(****************************************************************************************************************************************************)
(***********                           start of the controlling of the message overlay and blocking of the visualisation                             ************)
(****************************************************************************************************************************************************)
(* Activate Error Message Overlay *)
	IF xActiveErrorMsg AND NOT(xEmergency) AND NOT(xNoAirPressure) AND NOT(xNodeFailCANOpen) THEN
		CASE iStepFunction OF
		(* Check *)
		1:	T_StartUp.T_State.xBlockChangeMovementVisu:=TRUE;	(* Lock the navigation of the visu *)
			(* Overlay Message Error *)
			T_VisuQVis.ptrT_ExchgParam^.T_SafetyCtrl.bStateMessageError:=1;
			T_VisuQVis.ptrT_ExchgParam^.T_SafetyCtrl.bStateMessageInfo:=0;
			T_VisuQVis.ptrT_ExchgParam^.T_SafetyCtrl.bStateMessageWarning:=0;
			T_VisuQVis.ptrT_ExchgParam^.T_SafetyCtrl.iMsgErrorLine1:=iMsgNumber;
			T_VisuQVis.ptrT_ExchgParam^.T_SafetyCtrl.iMsgErrorLine2:=iMsgNumber;
			T_VisuQVis.ptrT_ExchgParam^.T_SafetyCtrl.iMsgErrorLine3:=iMsgNumber;
			T_VisuQVis.ptrT_ExchgParam^.T_SafetyCtrl.iMsgErrorLine4:=iMsgNumber;
			T_VisuQVis.ptrT_ExchgParam^.T_SafetyCtrl.xConfirmMsgError:=FALSE;
			T_VisuQVis.ptrT_ExchgParam^.T_SafetyCtrl.xBlockVisuObject:=TRUE;
			(* next step *)
			iStepFunction:=10;
		10:	IF T_VisuQVis.ptrT_ExchgParam^.T_SafetyCtrl.xConfirmMsgError THEN
				T_VisuQVis.ptrT_ExchgParam^.T_SafetyCtrl.xBlockVisuObject:=FALSE;
				T_StartUp.T_State.xBlockChangeMovementVisu:=FALSE;	(* Unlock the navigation of the visu *)
				T_VisuQVis.ptrT_ExchgParam^.T_SafetyCtrl.bStateMessageError:=0;
				T_VisuQVis.ptrT_ExchgParam^.T_SafetyCtrl.xConfirmMsgError:=FALSE;
				T_StartUp.T_Ctrle.xDone:=TRUE;
				T_StartUp.T_Ctrle.xErr:=FALSE;
				T_StartUp.T_Ctrle.udiErrorID:=16#0;
				xActiveErrorMsg:=FALSE;
				(* next step *)
				iStepFunction:=1;
			END_IF;
		END_CASE;
	END_IF;

(* Acitvate Info Message Overlay *)
	IF xActiveInfoMsg AND NOT(xEmergency) AND NOT(xNoAirPressure) AND NOT(xNodeFailCANOpen) THEN
		CASE iStepFunction OF
		(* Check *)
		1:	T_StartUp.T_State.xBlockChangeMovementVisu:=TRUE;	(* Lock the navigation of the visu *)
			(* Overlay Message Error *)
			T_VisuQVis.ptrT_ExchgParam^.T_SafetyCtrl.bStateMessageError:=0;
			T_VisuQVis.ptrT_ExchgParam^.T_SafetyCtrl.bStateMessageInfo:=1;
			T_VisuQVis.ptrT_ExchgParam^.T_SafetyCtrl.bStateMessageWarning:=0;
			T_VisuQVis.ptrT_ExchgParam^.T_SafetyCtrl.iMsgInfoLine1:=iMsgNumber;
			T_VisuQVis.ptrT_ExchgParam^.T_SafetyCtrl.iMsgInfoLine2:=iMsgNumber;
			T_VisuQVis.ptrT_ExchgParam^.T_SafetyCtrl.iMsgInfoLine3:=iMsgNumber;
			T_VisuQVis.ptrT_ExchgParam^.T_SafetyCtrl.iMsgInfoLine4:=iMsgNumber;
			T_VisuQVis.ptrT_ExchgParam^.T_SafetyCtrl.xConfirmMsgInfo:=FALSE;
			T_VisuQVis.ptrT_ExchgParam^.T_SafetyCtrl.xBlockVisuObject:=TRUE;
			(* next step *)
			iStepFunction:=10;
		10:	IF T_VisuQVis.ptrT_ExchgParam^.T_SafetyCtrl.xConfirmMsgInfo THEN
				T_VisuQVis.ptrT_ExchgParam^.T_SafetyCtrl.xBlockVisuObject:=FALSE;
				T_StartUp.T_State.xBlockChangeMovementVisu:=FALSE;	(* Unlock the navigation of the visu *)
				T_VisuQVis.ptrT_ExchgParam^.T_SafetyCtrl.bStateMessageInfo:=0;
				T_VisuQVis.ptrT_ExchgParam^.T_SafetyCtrl.xConfirmMsgInfo:=FALSE;
				T_StartUp.T_Ctrle.xDone:=TRUE;
				T_StartUp.T_Ctrle.xErr:=FALSE;
				T_StartUp.T_Ctrle.udiErrorID:=16#0;
				xActiveInfoMsg:=FALSE;
				(* next step *)
				iStepFunction:=1;
			END_IF;
		END_CASE;
	END_IF;
(****************************************************************************************************************************************************)
(***********                           end of the controlling of the message overlay and blocking of the visualisation                             ************)
(****************************************************************************************************************************************************)

	IF T_StartUp.T_Ctrle.xSetSecurityStateON THEN
		IF NOT(xReadFirstTime) THEN
			xReadFirstTime:=TRUE;
			iStepFunctionON:=1;
			TONWaitSetSecStateON(IN:=FALSE);
		END_IF;
		CASE iStepFunctionON OF
		1:	T_TwinSafeCtrleOUT.xTwinSAFE_Run:=FALSE;	(* Stop TwinSafe Groupe *)
			QarxDigitalOutput[1]:=FALSE;	(* QxCtrlLampStartButton *)
			QarxDigitalOutput[2]:=FALSE;	(* QxCtrlLampStopButton *)
			QarxDigitalOutput[3]:=FALSE;	(* QxCtrlLampReleaseButton *)
			TONWaitSetSecStateON(IN:=FALSE);
			iStepFunctionON:=2;
		2:	TONWaitSetSecStateON(IN:=TRUE,PT:=T#50ms);
			IF TONWaitSetSecStateON.Q THEN
				TONWaitSetSecStateON(IN:=FALSE);
				iStepFunctionON:=3;
			END_IF;
		3:	T_TwinSafeCtrleOUT.xTwinSAFE_Run:=TRUE;	(* Start TwinSafe Groupe *)
			T_StartUp.T_Ctrle.xSetSecurityStateON:=FALSE;
			xReadFirstTime:=FALSE;
			TONWaitSetSecStateON(IN:=FALSE);
			iStepFunctionON:=1;
		END_CASE;
	ELSE
		xReadFirstTime:=FALSE;
	END_IF;

(****************************************************************************************************************************************************)
(***********                   start of the execution of an emergeny stop, missing of air or an axis communication error                  ************)
(****************************************************************************************************************************************************)
(* Emergency or air supply *)
	IF xEmergency OR xNoAirPressure OR xNodeFailCANOpen THEN
		CASE iStepFunction OF
		1:	xSetOutputDisable:=TRUE;
			T_NovRAM.T_Ctrle.xReset:=TRUE;
			T_StartUp.T_State.xBlockChangeMovementVisu:=TRUE;
			T_StartUp.T_Ctrle.iMsgNumber:=0;
			T_VisuQVis.ptrT_ExchgParam^.T_SafetyCtrl.iStateStartPage:=0;	(* No Text *)
			T_VisuQVis.ptrT_ExchgParam^.T_Visu.T_Level.iPwSystem:=999;	(* Releas System Level *)
			T_VisuQVis.ptrT_ExchgParam^.T_Visu.T_Level.iActLevel:=1;
			T_Process.xError:=FALSE;
			IF T_Process.xEnable AND NOT(T_Process.xEnd) AND ((T_Process.iFunctNr >= 50) AND (T_Process.iFunctNr <= 53)) THEN
				(* Prozess ist aktiv und wurde unterbrochen, daher müssen die letzten änderungen an den InfoProzess Parameter in den NovRam abgespeichert werden *)
				(* next step *)
				iStepFunction:=2;
			ELSE
				IF xProcessAbordet THEN
					xProcessAbordet:=FALSE;
					(* next step *)
					iStepFunction:=2;
				ELSE
					(* next step *)
					iStepFunction:=3;
				END_IF;
			END_IF;
		2:	IF NOT(T_NovRAM.T_Ctrle.xReset) AND T_NovRAM.T_Ctrle.xDone THEN
				iStepFunction:=3;
			END_IF;
		3:	IF NOT(T_NovRAM.T_Ctrle.xReset) AND T_NovRAM.T_Ctrle.xDone THEN
				T_VisuQVis.T_CtrleVisu.xReset:=TRUE;
				iStepFunction:=10;
			END_IF;
		(* waiting confirm *)
		10:	IF NOT(xSetOutputDisable) AND NOT(T_VisuQVis.T_CtrleVisu.xReset) THEN
				IF xNoAirPressure THEN
					(* next step *)
					iStepFunction:=60;
				END_IF;
				IF xEmergency THEN
					(* next step *)
					iStepFunction:=20;
				END_IF;
				IF xNodeFailCANOpen THEN
					(* next step *)
					iStepFunction:=80;
				END_IF;
			END_IF
		20:	(* Overlay Message Error *)
			T_VisuQVis.ptrT_ExchgParam^.T_SafetyCtrl.bStateMessageError:=1;
			T_VisuQVis.ptrT_ExchgParam^.T_SafetyCtrl.bStateMessageInfo:=0;
			T_VisuQVis.ptrT_ExchgParam^.T_SafetyCtrl.bStateMessageWarning:=0;
			T_VisuQVis.ptrT_ExchgParam^.T_SafetyCtrl.iMsgErrorLine1:=1;	(* EMERGENCY STOP BUTTON IS ACITVE! *)
			T_VisuQVis.ptrT_ExchgParam^.T_SafetyCtrl.iMsgErrorLine2:=1;	(* PLEASE RELEASE THIS BUTTON *)
			T_VisuQVis.ptrT_ExchgParam^.T_SafetyCtrl.iMsgErrorLine3:=1;	(* AND AFTER CONFIRM THIS MESSAGE *)
			T_VisuQVis.ptrT_ExchgParam^.T_SafetyCtrl.iMsgErrorLine4:=1;	(*  *)
			T_VisuQVis.ptrT_ExchgParam^.T_SafetyCtrl.xConfirmMsgError:=FALSE;
			T_VisuQVis.ptrT_ExchgParam^.T_SafetyCtrl.xBlockVisuObject:=TRUE;
			(* next step *)
			iStepFunction:=30;
		30:	IF T_VisuQVis.ptrT_ExchgParam^.T_SafetyCtrl.xConfirmMsgError THEN
				T_VisuQVis.ptrT_ExchgParam^.T_SafetyCtrl.xBlockVisuObject:=FALSE;
				T_VisuQVis.ptrT_ExchgParam^.T_SafetyCtrl.bStateMessageError:=0;
				T_VisuQVis.ptrT_ExchgParam^.T_SafetyCtrl.xConfirmMsgError:=FALSE;
				IF NOT(T_TwinSafeIn.IxEmergencyStopMachine) OR NOT(T_TwinSafeIn.IxEmergencyStopStuder) THEN
					(* next step *)
					iStepFunction:=20;
				ELSE
					(* next step *)
					iStepFunction:=90;
				END_IF;
			END_IF;
		60:	(* Overlay Message Error *)
			T_VisuQVis.ptrT_ExchgParam^.T_SafetyCtrl.bStateMessageError:=1;
			T_VisuQVis.ptrT_ExchgParam^.T_SafetyCtrl.bStateMessageInfo:=0;
			T_VisuQVis.ptrT_ExchgParam^.T_SafetyCtrl.bStateMessageWarning:=0;
			T_VisuQVis.ptrT_ExchgParam^.T_SafetyCtrl.iMsgErrorLine1:=2;	(* NO AIR PRESSURE! *)
			T_VisuQVis.ptrT_ExchgParam^.T_SafetyCtrl.iMsgErrorLine2:=2;	(* PLEASE ACTIVATE THE AIR PRESSURE *)
			T_VisuQVis.ptrT_ExchgParam^.T_SafetyCtrl.iMsgErrorLine3:=2;	(* AND AFTER CONFIRM THIS MESSAGE *)
			T_VisuQVis.ptrT_ExchgParam^.T_SafetyCtrl.iMsgErrorLine4:=2;	(*  *)
			T_VisuQVis.ptrT_ExchgParam^.T_SafetyCtrl.xConfirmMsgError:=FALSE;
			T_VisuQVis.ptrT_ExchgParam^.T_SafetyCtrl.xBlockVisuObject:=TRUE;
			FBErrorMessage(	diErrorNr:=7,		(* No Air Pressure *)
							T_ErrorList:=T_ErrorList);
			T_VisuQVis.ptrT_ExchgParam^.T_Visu.T_Message.sDynamicTextEnglish:=FBErrorMessage.sErrorTextEnglish;
			T_VisuQVis.ptrT_ExchgParam^.T_Visu.T_Message.sDynamicTextDeutsch:=FBErrorMessage.sErrorTextDeutsch;
			T_VisuQVis.ptrT_ExchgParam^.T_Visu.T_Message.sDynamicTextFrancais:=FBErrorMessage.sErrorTextFrancais;
			(* Safe the error *)
			T_VisuQVis.ptrT_ExchgParam^.T_SafetyCtrl.diSetForceErrorNr:=7;
			T_VisuQVis.ptrT_ExchgParam^.T_SafetyCtrl.xSetForceError:=TRUE;
			(* next step *)
			iStepFunction:=70;
		70:	IF T_VisuQVis.ptrT_ExchgParam^.T_SafetyCtrl.xConfirmMsgError THEN
				T_VisuQVis.ptrT_ExchgParam^.T_SafetyCtrl.xBlockVisuObject:=FALSE;
				T_VisuQVis.ptrT_ExchgParam^.T_SafetyCtrl.bStateMessageError:=0;
				T_VisuQVis.ptrT_ExchgParam^.T_SafetyCtrl.xConfirmMsgError:=FALSE;
				(* next step *)
				iStepFunction:=90;
			END_IF;
		80:	(* Overlay Message Error *)
			T_VisuQVis.ptrT_ExchgParam^.T_SafetyCtrl.bStateMessageError:=1;
			T_VisuQVis.ptrT_ExchgParam^.T_SafetyCtrl.bStateMessageInfo:=0;
			T_VisuQVis.ptrT_ExchgParam^.T_SafetyCtrl.bStateMessageWarning:=0;
			T_VisuQVis.ptrT_ExchgParam^.T_SafetyCtrl.iMsgErrorLine1:=21;	(* AT LEAST ONE CANOPEN CONTROLLER FAILED! *)
			T_VisuQVis.ptrT_ExchgParam^.T_SafetyCtrl.iMsgErrorLine2:=21;	(* PLEASE CHECK THE ECOSTEP AXIS *)
			T_VisuQVis.ptrT_ExchgParam^.T_SafetyCtrl.iMsgErrorLine3:=21;	(* AND CONFIRM THIS MESSAGE *)
			T_VisuQVis.ptrT_ExchgParam^.T_SafetyCtrl.iMsgErrorLine4:=21;	(*  *)
			T_VisuQVis.ptrT_ExchgParam^.T_SafetyCtrl.xConfirmMsgError:=FALSE;
			T_VisuQVis.ptrT_ExchgParam^.T_SafetyCtrl.xBlockVisuObject:=TRUE;
			FBErrorMessage(	diErrorNr:=6,		(* At least one Ecostep CANOpen Controller failed! *)
							T_ErrorList:=T_ErrorList);
			T_VisuQVis.ptrT_ExchgParam^.T_Visu.T_Message.sDynamicTextEnglish:=FBErrorMessage.sErrorTextEnglish;
			T_VisuQVis.ptrT_ExchgParam^.T_Visu.T_Message.sDynamicTextDeutsch:=FBErrorMessage.sErrorTextDeutsch;
			T_VisuQVis.ptrT_ExchgParam^.T_Visu.T_Message.sDynamicTextFrancais:=FBErrorMessage.sErrorTextFrancais;
			(* Safe the error *)
			T_VisuQVis.ptrT_ExchgParam^.T_SafetyCtrl.diSetForceErrorNr:=6;
			T_VisuQVis.ptrT_ExchgParam^.T_SafetyCtrl.xSetForceError:=TRUE;
			(* next step *)
			iStepFunction:=81;
		81:	IF T_VisuQVis.ptrT_ExchgParam^.T_SafetyCtrl.xConfirmMsgError THEN
				T_VisuQVis.ptrT_ExchgParam^.T_SafetyCtrl.xBlockVisuObject:=FALSE;
				T_VisuQVis.ptrT_ExchgParam^.T_SafetyCtrl.bStateMessageError:=0;
				T_VisuQVis.ptrT_ExchgParam^.T_SafetyCtrl.xConfirmMsgError:=FALSE;
				(* next step *)
				iStepFunction:=90;
			END_IF;
		(* end function or time out *)
		90:	xActiveErrorMsg:=FALSE;
			xActiveInfoMsg:=FALSE;
			T_StartUp.T_Ctrle.xDone:=TRUE;
			T_StartUp.T_Ctrle.xErr:=FALSE;
			T_StartUp.T_Ctrle.udiErrorID:=0;
			xEmergency:=FALSE;
			xNoAirPressure:=FALSE;
			xNodeFailCANOpen:=FALSE;
			xStartBooting:=TRUE;
			tTimeOutFunction:=T#0s;	(* deactivate the time out *)
			(* next step *)
			iStepFunction:=1;
		END_CASE
	END_IF;
(****************************************************************************************************************************************************)
(***********                   start of the execution of an emergeny stop, missing of air or an axis communication error                  ************)
(****************************************************************************************************************************************************)

(* Delete of the line error message *)
	IF xDeleteErrorMessage THEN
		xDeleteErrorMessage:=FALSE;
		FBInitErrorList(T_ErrorList:= T_ErrorList);	(* Init Static Text for Error List *)
		T_VisuQVis.ptrT_ExchgParam^.T_Visu.T_Message.sDynamicTextEnglish:='';
		T_VisuQVis.ptrT_ExchgParam^.T_Visu.T_Message.sDynamicTextDeutsch:='';
		T_VisuQVis.ptrT_ExchgParam^.T_Visu.T_Message.sDynamicTextFrancais:='';
		T_VisuQVis.ptrT_ExchgParam^.T_Visu.T_Message.iState:=0;
	END_IF;

(* Set Output disabled *)
	IF xSetOutputDisable THEN
		T_TwinSafeCtrleOUT.xTwinSAFE_Run:=FALSE;	(* Stop TwinSafe Groupe *)
		T_Process.xEnable:=FALSE;
		QarxDigitalOutput[1]:=FALSE;	(* QxCtrlLampStartButton *)
		QarxDigitalOutput[2]:=FALSE;	(* QxCtrlLampStopButton *)
		QarxDigitalOutput[3]:=FALSE;	(* QxCtrlLampReleaseButton *)
		QarxDigitalOutput[4]:=FALSE;	(* QxCtrlLampCurEcoButton *)
		T_Station.TControl.xEnable:=FALSE;
		T_VisuQVis.ptrT_ExchgParam^.T_Visu.iLoadingStartPage:=1;
		(* confirm *)
		xSetOutputDisable:=FALSE;
	END_IF
END_PROGRAM

(* POU PRG_PROCESS_LAYER4/FB_PROCESS/FB_InitErrorList, ST *)
FUNCTION_BLOCK FB_InitErrorList
VAR_INPUT
END_VAR
VAR_IN_OUT
	T_ErrorList:ST_ERROR_LIST;
END_VAR
VAR_OUTPUT
END_VAR
VAR
END_VAR
(****************************************************************************************************************************************************)
(***********                                    This Functionblock init all the error text in english, german and french                                       ************)
(****************************************************************************************************************************************************)
(* Static English Error List *)
T_ErrorList.asErrorListEnglish.T_LanguagList[1]:='Internal problem, should never appear';
T_ErrorList.asErrorListEnglish.T_LanguagList[2]:='Antivalence error of the motor encoder';
T_ErrorList.asErrorListEnglish.T_LanguagList[3]:='Encoder counter error, >+/- 4 inc';
T_ErrorList.asErrorListEnglish.T_LanguagList[4]:='Mster encoder X7 counter error, >+/- 4 inc';
T_ErrorList.asErrorListEnglish.T_LanguagList[5]:='Heat sink temperature to high (>80°)';
T_ErrorList.asErrorListEnglish.T_LanguagList[6]:='Low voltage (<18V) of the +24V logic supply';
T_ErrorList.asErrorListEnglish.T_LanguagList[7]:='High voltage X10 (>180V) of the motor power supply';
T_ErrorList.asErrorListEnglish.T_LanguagList[8]:='Low voltage X10 (<24V) of the motor power supply';
T_ErrorList.asErrorListEnglish.T_LanguagList[9]:='Short circuit in the motor phase A';
T_ErrorList.asErrorListEnglish.T_LanguagList[10]:='Short circuit in the motor phase B';
T_ErrorList.asErrorListEnglish.T_LanguagList[11]:='Short circuit of a digital output';
T_ErrorList.asErrorListEnglish.T_LanguagList[12]:='Digital input ENABLE going to low level';
T_ErrorList.asErrorListEnglish.T_LanguagList[13]:='Exceed max. countouring error';
T_ErrorList.asErrorListEnglish.T_LanguagList[14]:='Rotation speed to high, can not read encoder signal';
T_ErrorList.asErrorListEnglish.T_LanguagList[15]:='Can not find the commutation';
T_ErrorList.asErrorListEnglish.T_LanguagList[16]:='CAN-Communication broken by Node Guarding';
T_ErrorList.asErrorListEnglish.T_LanguagList[17]:='I^2t- Controlling triggered (current limit)';
T_ErrorList.asErrorListEnglish.T_LanguagList[18]:='ADS communication error';
T_ErrorList.asErrorListEnglish.T_LanguagList[19]:='Axis function time out error';
T_ErrorList.asErrorListEnglish.T_LanguagList[20]:='Axis function not implemented';
T_ErrorList.asErrorListEnglish.T_LanguagList[21]:='No HDD free resource, time out';
T_ErrorList.asErrorListEnglish.T_LanguagList[22]:='HDD error, no file found';
T_ErrorList.asErrorListEnglish.T_LanguagList[23]:='Axis Parameter File, wrong syntax';
T_ErrorList.asErrorListEnglish.T_LanguagList[24]:='Wrong Para Fct: Read Axis Parameter';
T_ErrorList.asErrorListEnglish.T_LanguagList[25]:='Limit End Switch Active';
T_ErrorList.asErrorListEnglish.T_LanguagList[26]:='PDOMapping Para File, wrong syntax';
T_ErrorList.asErrorListEnglish.T_LanguagList[27]:='Wrong Para Fct: Read PDOMapping Parameter';
T_ErrorList.asErrorListEnglish.T_LanguagList[28]:='No Axis Power Supply';
T_ErrorList.asErrorListEnglish.T_LanguagList[29]:='Wrong Para Fct: Move velocity';
T_ErrorList.asErrorListEnglish.T_LanguagList[30]:='Can not move, no power supply';
T_ErrorList.asErrorListEnglish.T_LanguagList[31]:='Wrong Para Fct: Move position absolute';
T_ErrorList.asErrorListEnglish.T_LanguagList[32]:='Wrong Para Fct: Move position relative';
T_ErrorList.asErrorListEnglish.T_LanguagList[33]:='Wrong Para Fct: Move referencing';
T_ErrorList.asErrorListEnglish.T_LanguagList[34]:='Fct CalcAnlgeRefIndex:Ref.Sensor not found';
T_ErrorList.asErrorListEnglish.T_LanguagList[35]:='Wrong Para Fct: Send Axis Parameter';
T_ErrorList.asErrorListEnglish.T_LanguagList[36]:='Wrong Para Fct: Send PDOMapping Parameter';
T_ErrorList.asErrorListEnglish.T_LanguagList[37]:='Wrong Para Fct: Master/Slave';
T_ErrorList.asErrorListEnglish.T_LanguagList[38]:='Axis general error';
T_ErrorList.asErrorListEnglish.T_LanguagList[39]:='ToolLeft: Wrong configuration or Axis missing';
T_ErrorList.asErrorListEnglish.T_LanguagList[40]:='ToolCenter: Wrong configuration or Axis missing';
T_ErrorList.asErrorListEnglish.T_LanguagList[41]:='ToolRight: Wrong configuration or Axis missing';
T_ErrorList.asErrorListEnglish.T_LanguagList[42]:='ToolFeeder: Wrong configuration or Axis missing';
T_ErrorList.asErrorListEnglish.T_LanguagList[43]:='GrindFeeder: Wrong configuration or Axis missing';
T_ErrorList.asErrorListEnglish.T_LanguagList[44]:='BoxId general error';
T_ErrorList.asErrorListEnglish.T_LanguagList[45]:='Cyl. Function not implemented';
T_ErrorList.asErrorListEnglish.T_LanguagList[46]:='Sensor down not active';
T_ErrorList.asErrorListEnglish.T_LanguagList[47]:='Sensor up not active';
T_ErrorList.asErrorListEnglish.T_LanguagList[48]:='Cyl. general error';
T_ErrorList.asErrorListEnglish.T_LanguagList[49]:='File for profile not found';
T_ErrorList.asErrorListEnglish.T_LanguagList[50]:='Profile file not found: ';
T_ErrorList.asErrorListEnglish.T_LanguagList[51]:='--> Load static default parameter';
T_ErrorList.asErrorListEnglish.T_LanguagList[52]:='Machine is not referenced';
T_ErrorList.asErrorListEnglish.T_LanguagList[53]:='Settled parameter for ToolLength is to long';
T_ErrorList.asErrorListEnglish.T_LanguagList[54]:='Settled parameter for ToolLength is to short';
T_ErrorList.asErrorListEnglish.T_LanguagList[55]:='Settled parameter for ToolDiameter is to big';
T_ErrorList.asErrorListEnglish.T_LanguagList[56]:='Settled parameter for ToolDiameter is to small';
T_ErrorList.asErrorListEnglish.T_LanguagList[57]:='Tool is not clamped';
T_ErrorList.asErrorListEnglish.T_LanguagList[58]:='ToolTension is not active';
T_ErrorList.asErrorListEnglish.T_LanguagList[59]:='ToolFeeeder is not on the StartPosition';
T_ErrorList.asErrorListEnglish.T_LanguagList[60]:='At least one Axis is busy';
T_ErrorList.asErrorListEnglish.T_LanguagList[61]:='Undefined Station error';
T_ErrorList.asErrorListEnglish.T_LanguagList[62]:='At least a passage of a section is not equal';
T_ErrorList.asErrorListEnglish.T_LanguagList[63]:='On the MicroWire it is not possible to Referencing';
T_ErrorList.asErrorListEnglish.T_LanguagList[64]:='Undefined Machine Error';
T_ErrorList.asErrorListEnglish.T_LanguagList[65]:='At least one Ecostep CANOpen Controller failed!';
T_ErrorList.asErrorListEnglish.T_LanguagList[66]:='No Air Pressure';
T_ErrorList.asErrorListEnglish.T_LanguagList[67]:='At least one settled diameter is bigger than ToolDiameter';
T_ErrorList.asErrorListEnglish.T_LanguagList[68]:='ToolTension is active';
T_ErrorList.asErrorListEnglish.T_LanguagList[69]:='';
T_ErrorList.asErrorListEnglish.T_LanguagList[70]:='';
T_ErrorList.asErrorListEnglish.T_LanguagList[71]:='';
T_ErrorList.asErrorListEnglish.T_LanguagList[72]:='';
T_ErrorList.asErrorListEnglish.T_LanguagList[73]:='';
T_ErrorList.asErrorListEnglish.T_LanguagList[74]:='';
T_ErrorList.asErrorListEnglish.T_LanguagList[75]:='';
T_ErrorList.asErrorListEnglish.T_LanguagList[76]:='';
T_ErrorList.asErrorListEnglish.T_LanguagList[77]:='';
T_ErrorList.asErrorListEnglish.T_LanguagList[78]:='';
T_ErrorList.asErrorListEnglish.T_LanguagList[79]:='';
T_ErrorList.asErrorListEnglish.T_LanguagList[80]:='';
T_ErrorList.asErrorListEnglish.T_LanguagList[81]:='';
T_ErrorList.asErrorListEnglish.T_LanguagList[82]:='';
T_ErrorList.asErrorListEnglish.T_LanguagList[83]:='';
T_ErrorList.asErrorListEnglish.T_LanguagList[84]:='';
T_ErrorList.asErrorListEnglish.T_LanguagList[85]:='';
T_ErrorList.asErrorListEnglish.T_LanguagList[86]:='';
T_ErrorList.asErrorListEnglish.T_LanguagList[87]:='';
T_ErrorList.asErrorListEnglish.T_LanguagList[88]:='';
T_ErrorList.asErrorListEnglish.T_LanguagList[89]:='';
T_ErrorList.asErrorListEnglish.T_LanguagList[90]:='';
T_ErrorList.asErrorListEnglish.T_LanguagList[91]:='';
T_ErrorList.asErrorListEnglish.T_LanguagList[92]:='';
T_ErrorList.asErrorListEnglish.T_LanguagList[93]:='';
T_ErrorList.asErrorListEnglish.T_LanguagList[94]:='';
T_ErrorList.asErrorListEnglish.T_LanguagList[95]:='';
T_ErrorList.asErrorListEnglish.T_LanguagList[96]:='';
T_ErrorList.asErrorListEnglish.T_LanguagList[97]:='';
T_ErrorList.asErrorListEnglish.T_LanguagList[98]:='';
T_ErrorList.asErrorListEnglish.T_LanguagList[99]:='';
T_ErrorList.asErrorListEnglish.T_LanguagList[100]:='';
T_ErrorList.asErrorListEnglish.T_LanguagList[101]:='';
T_ErrorList.asErrorListEnglish.T_LanguagList[102]:='';
T_ErrorList.asErrorListEnglish.T_LanguagList[103]:='';
T_ErrorList.asErrorListEnglish.T_LanguagList[104]:='';
T_ErrorList.asErrorListEnglish.T_LanguagList[105]:='';
T_ErrorList.asErrorListEnglish.T_LanguagList[106]:='';
T_ErrorList.asErrorListEnglish.T_LanguagList[107]:='';
T_ErrorList.asErrorListEnglish.T_LanguagList[108]:='';
T_ErrorList.asErrorListEnglish.T_LanguagList[109]:='';
T_ErrorList.asErrorListEnglish.T_LanguagList[110]:='';
T_ErrorList.asErrorListEnglish.T_LanguagList[111]:='';
T_ErrorList.asErrorListEnglish.T_LanguagList[112]:='';
T_ErrorList.asErrorListEnglish.T_LanguagList[113]:='';
T_ErrorList.asErrorListEnglish.T_LanguagList[114]:='';
T_ErrorList.asErrorListEnglish.T_LanguagList[115]:='';
T_ErrorList.asErrorListEnglish.T_LanguagList[116]:='';
T_ErrorList.asErrorListEnglish.T_LanguagList[117]:='';
T_ErrorList.asErrorListEnglish.T_LanguagList[118]:='';
T_ErrorList.asErrorListEnglish.T_LanguagList[119]:='';
T_ErrorList.asErrorListEnglish.T_LanguagList[120]:='';
T_ErrorList.asErrorListEnglish.T_LanguagList[121]:='';
T_ErrorList.asErrorListEnglish.T_LanguagList[122]:='';
T_ErrorList.asErrorListEnglish.T_LanguagList[123]:='';
T_ErrorList.asErrorListEnglish.T_LanguagList[124]:='';
T_ErrorList.asErrorListEnglish.T_LanguagList[125]:='';
T_ErrorList.asErrorListEnglish.T_LanguagList[126]:='';
T_ErrorList.asErrorListEnglish.T_LanguagList[127]:='';
T_ErrorList.asErrorListEnglish.T_LanguagList[128]:='';
T_ErrorList.asErrorListEnglish.T_LanguagList[129]:='';
T_ErrorList.asErrorListEnglish.T_LanguagList[130]:='';
T_ErrorList.asErrorListEnglish.T_LanguagList[131]:='';
T_ErrorList.asErrorListEnglish.T_LanguagList[132]:='';
T_ErrorList.asErrorListEnglish.T_LanguagList[133]:='';
T_ErrorList.asErrorListEnglish.T_LanguagList[134]:='';
T_ErrorList.asErrorListEnglish.T_LanguagList[135]:='';
T_ErrorList.asErrorListEnglish.T_LanguagList[136]:='';
T_ErrorList.asErrorListEnglish.T_LanguagList[137]:='';
T_ErrorList.asErrorListEnglish.T_LanguagList[138]:='';
T_ErrorList.asErrorListEnglish.T_LanguagList[139]:='';
T_ErrorList.asErrorListEnglish.T_LanguagList[140]:='';
T_ErrorList.asErrorListEnglish.T_LanguagList[141]:='';
T_ErrorList.asErrorListEnglish.T_LanguagList[142]:='';
T_ErrorList.asErrorListEnglish.T_LanguagList[143]:='';
T_ErrorList.asErrorListEnglish.T_LanguagList[144]:='';
T_ErrorList.asErrorListEnglish.T_LanguagList[145]:='';
T_ErrorList.asErrorListEnglish.T_LanguagList[146]:='';
T_ErrorList.asErrorListEnglish.T_LanguagList[147]:='';
T_ErrorList.asErrorListEnglish.T_LanguagList[148]:='';
T_ErrorList.asErrorListEnglish.T_LanguagList[149]:='';
T_ErrorList.asErrorListEnglish.T_LanguagList[150]:='';
T_ErrorList.asErrorListEnglish.T_LanguagList[151]:='';
T_ErrorList.asErrorListEnglish.T_LanguagList[152]:='';
T_ErrorList.asErrorListEnglish.T_LanguagList[153]:='';
T_ErrorList.asErrorListEnglish.T_LanguagList[154]:='';
T_ErrorList.asErrorListEnglish.T_LanguagList[155]:='';
T_ErrorList.asErrorListEnglish.T_LanguagList[156]:='';
T_ErrorList.asErrorListEnglish.T_LanguagList[157]:='';
T_ErrorList.asErrorListEnglish.T_LanguagList[158]:='';
T_ErrorList.asErrorListEnglish.T_LanguagList[159]:='';
T_ErrorList.asErrorListEnglish.T_LanguagList[160]:='';
T_ErrorList.asErrorListEnglish.T_LanguagList[161]:='';
T_ErrorList.asErrorListEnglish.T_LanguagList[162]:='';
T_ErrorList.asErrorListEnglish.T_LanguagList[163]:='';
T_ErrorList.asErrorListEnglish.T_LanguagList[164]:='';
T_ErrorList.asErrorListEnglish.T_LanguagList[165]:='';
T_ErrorList.asErrorListEnglish.T_LanguagList[166]:='';
T_ErrorList.asErrorListEnglish.T_LanguagList[167]:='';
T_ErrorList.asErrorListEnglish.T_LanguagList[168]:='';
T_ErrorList.asErrorListEnglish.T_LanguagList[169]:='';
T_ErrorList.asErrorListEnglish.T_LanguagList[170]:='';
T_ErrorList.asErrorListEnglish.T_LanguagList[171]:='';
T_ErrorList.asErrorListEnglish.T_LanguagList[172]:='';

(* Static Deutsch Error List *)
T_ErrorList.asErrorListDeutsch.T_LanguagList[1]:='Interne Ursache, darf niemals auftreten';
T_ErrorList.asErrorListDeutsch.T_LanguagList[2]:='Antivalenzfehler der Motorencodersignale';
T_ErrorList.asErrorListDeutsch.T_LanguagList[3]:='Encoder Zählfehler, >+/- 4 ink';
T_ErrorList.asErrorListDeutsch.T_LanguagList[4]:='Master Encoder X7 Zählfehler, >+/- 4 inc';
T_ErrorList.asErrorListDeutsch.T_LanguagList[5]:='Kühlkörpertemperatur zu hoch (> 80°)';
T_ErrorList.asErrorListDeutsch.T_LanguagList[6]:='Unterspannung (<18V) der +24V Logikversorgung';
T_ErrorList.asErrorListDeutsch.T_LanguagList[7]:='Überspannung X10 (>180V) der Leistungsversorgung';
T_ErrorList.asErrorListDeutsch.T_LanguagList[8]:='Unterspannung X10 (<24V) der Leistungsversorgung';
T_ErrorList.asErrorListDeutsch.T_LanguagList[9]:='Kurzschluss in Motorphase A';
T_ErrorList.asErrorListDeutsch.T_LanguagList[10]:='Kurzschluss in Motorphase B';
T_ErrorList.asErrorListDeutsch.T_LanguagList[11]:='Kurzschluss eines digitalen Ausgangs';
T_ErrorList.asErrorListDeutsch.T_LanguagList[12]:='Digital-Eingang ENABLE wurde auf Low-Pegel gesetzt';
T_ErrorList.asErrorListDeutsch.T_LanguagList[13]:='Max. Schleppfehler überschritten';
T_ErrorList.asErrorListDeutsch.T_LanguagList[14]:='Drehzahl zu hoch, Regler kann Encoder nicht mehr auslesen';
T_ErrorList.asErrorListDeutsch.T_LanguagList[15]:='Kommutierung nicht gefunden';
T_ErrorList.asErrorListDeutsch.T_LanguagList[16]:='CAN-Kommunikation unterbrochen bei Node Guarding';
T_ErrorList.asErrorListDeutsch.T_LanguagList[17]:='I^2t- Überwachung ausgelöst (Stromgrenze)';
T_ErrorList.asErrorListDeutsch.T_LanguagList[18]:='ADS communication error';
T_ErrorList.asErrorListDeutsch.T_LanguagList[19]:='Axis function time out error';
T_ErrorList.asErrorListDeutsch.T_LanguagList[20]:='Axis function not implemented';
T_ErrorList.asErrorListDeutsch.T_LanguagList[21]:='No HDD free resource, time out';
T_ErrorList.asErrorListDeutsch.T_LanguagList[22]:='HDD error, no file found';
T_ErrorList.asErrorListDeutsch.T_LanguagList[23]:='Axis Parameter File, wrong syntax';
T_ErrorList.asErrorListDeutsch.T_LanguagList[24]:='Wrong Para Fct: Read Axis Parameter';
T_ErrorList.asErrorListDeutsch.T_LanguagList[25]:='Limit End Switch Active';
T_ErrorList.asErrorListDeutsch.T_LanguagList[26]:='PDOMapping Para File, wrong syntax';
T_ErrorList.asErrorListDeutsch.T_LanguagList[27]:='Wrong Para Fct: Read PDOMapping Parameter';
T_ErrorList.asErrorListDeutsch.T_LanguagList[28]:='No Axis Power Supply';
T_ErrorList.asErrorListDeutsch.T_LanguagList[29]:='Wrong Para Fct: Move velocity';
T_ErrorList.asErrorListDeutsch.T_LanguagList[30]:='Can not move, no power supply';
T_ErrorList.asErrorListDeutsch.T_LanguagList[31]:='Wrong Para Fct: Move position absolute';
T_ErrorList.asErrorListDeutsch.T_LanguagList[32]:='Wrong Para Fct: Move position relative';
T_ErrorList.asErrorListDeutsch.T_LanguagList[33]:='Wrong Para Fct: Move referencing';
T_ErrorList.asErrorListDeutsch.T_LanguagList[34]:='Fct CalcAnlgeRefIndex:Ref.Sensor not found';
T_ErrorList.asErrorListDeutsch.T_LanguagList[35]:='Wrong Para Fct: Send Axis Parameter';
T_ErrorList.asErrorListDeutsch.T_LanguagList[36]:='Wrong Para Fct: Send PDOMapping Parameter';
T_ErrorList.asErrorListDeutsch.T_LanguagList[37]:='Wrong Para Fct: Master/Slave';
T_ErrorList.asErrorListDeutsch.T_LanguagList[38]:='Axis general error';
T_ErrorList.asErrorListDeutsch.T_LanguagList[39]:='ToolLeft: Wrong configuration or Axis missing';
T_ErrorList.asErrorListDeutsch.T_LanguagList[40]:='ToolCenter: Wrong configuration or Axis missing';
T_ErrorList.asErrorListDeutsch.T_LanguagList[41]:='ToolRight: Wrong configuration or Axis missing';
T_ErrorList.asErrorListDeutsch.T_LanguagList[42]:='ToolFeeder: Wrong configuration or Axis missing';
T_ErrorList.asErrorListDeutsch.T_LanguagList[43]:='GrindFeeder: Wrong configuration or Axis missing';
T_ErrorList.asErrorListDeutsch.T_LanguagList[44]:='BoxId general error';
T_ErrorList.asErrorListDeutsch.T_LanguagList[45]:='Cyl. Function not implemented';
T_ErrorList.asErrorListDeutsch.T_LanguagList[46]:='Sensor down not active';
T_ErrorList.asErrorListDeutsch.T_LanguagList[47]:='Sensor up not active';
T_ErrorList.asErrorListDeutsch.T_LanguagList[48]:='Cyl. general error';
T_ErrorList.asErrorListDeutsch.T_LanguagList[49]:='File for profile not found';
T_ErrorList.asErrorListDeutsch.T_LanguagList[50]:='Profile file not found: ';
T_ErrorList.asErrorListDeutsch.T_LanguagList[51]:='--> Load static default parameter';
T_ErrorList.asErrorListDeutsch.T_LanguagList[52]:='Machine is not referenced';
T_ErrorList.asErrorListDeutsch.T_LanguagList[53]:='Settled parameter for ToolLength is to long';
T_ErrorList.asErrorListDeutsch.T_LanguagList[54]:='Settled parameter for ToolLength is to short';
T_ErrorList.asErrorListDeutsch.T_LanguagList[55]:='Settled parameter for ToolDiameter is to big';
T_ErrorList.asErrorListDeutsch.T_LanguagList[56]:='Settled parameter for ToolDiameter is to small';
T_ErrorList.asErrorListDeutsch.T_LanguagList[57]:='Tool is not clamped';
T_ErrorList.asErrorListDeutsch.T_LanguagList[58]:='ToolTension is not active';
T_ErrorList.asErrorListDeutsch.T_LanguagList[59]:='ToolFeeeder is not on the StartPosition';
T_ErrorList.asErrorListDeutsch.T_LanguagList[60]:='At least one Axis is busy';
T_ErrorList.asErrorListDeutsch.T_LanguagList[61]:='Undefined Station error';
T_ErrorList.asErrorListDeutsch.T_LanguagList[62]:='At least a passage of a section is not equal';
T_ErrorList.asErrorListDeutsch.T_LanguagList[63]:='On the MicroWire it is not possible to Referencing';
T_ErrorList.asErrorListDeutsch.T_LanguagList[64]:='Undefined Machine Error';
T_ErrorList.asErrorListDeutsch.T_LanguagList[65]:='At least one Ecostep CANOpen Controller failed!';
T_ErrorList.asErrorListDeutsch.T_LanguagList[66]:='No Air Pressure';
T_ErrorList.asErrorListDeutsch.T_LanguagList[67]:='At least one settled diameter is bigger than ToolDiameter';
T_ErrorList.asErrorListDeutsch.T_LanguagList[68]:='ToolTension is active';
T_ErrorList.asErrorListDeutsch.T_LanguagList[69]:='';
T_ErrorList.asErrorListDeutsch.T_LanguagList[70]:='';
T_ErrorList.asErrorListDeutsch.T_LanguagList[71]:='';
T_ErrorList.asErrorListDeutsch.T_LanguagList[72]:='';
T_ErrorList.asErrorListDeutsch.T_LanguagList[73]:='';
T_ErrorList.asErrorListDeutsch.T_LanguagList[74]:='';
T_ErrorList.asErrorListDeutsch.T_LanguagList[75]:='';
T_ErrorList.asErrorListDeutsch.T_LanguagList[76]:='';
T_ErrorList.asErrorListDeutsch.T_LanguagList[77]:='';
T_ErrorList.asErrorListDeutsch.T_LanguagList[78]:='';
T_ErrorList.asErrorListDeutsch.T_LanguagList[79]:='';
T_ErrorList.asErrorListDeutsch.T_LanguagList[80]:='';
T_ErrorList.asErrorListDeutsch.T_LanguagList[81]:='';
T_ErrorList.asErrorListDeutsch.T_LanguagList[82]:='';
T_ErrorList.asErrorListDeutsch.T_LanguagList[83]:='';
T_ErrorList.asErrorListDeutsch.T_LanguagList[84]:='';
T_ErrorList.asErrorListDeutsch.T_LanguagList[85]:='';
T_ErrorList.asErrorListDeutsch.T_LanguagList[86]:='';
T_ErrorList.asErrorListDeutsch.T_LanguagList[87]:='';
T_ErrorList.asErrorListDeutsch.T_LanguagList[88]:='';
T_ErrorList.asErrorListDeutsch.T_LanguagList[89]:='';
T_ErrorList.asErrorListDeutsch.T_LanguagList[90]:='';
T_ErrorList.asErrorListDeutsch.T_LanguagList[91]:='';
T_ErrorList.asErrorListDeutsch.T_LanguagList[92]:='';
T_ErrorList.asErrorListDeutsch.T_LanguagList[93]:='';
T_ErrorList.asErrorListDeutsch.T_LanguagList[94]:='';
T_ErrorList.asErrorListDeutsch.T_LanguagList[95]:='';
T_ErrorList.asErrorListDeutsch.T_LanguagList[96]:='';
T_ErrorList.asErrorListDeutsch.T_LanguagList[97]:='';
T_ErrorList.asErrorListDeutsch.T_LanguagList[98]:='';
T_ErrorList.asErrorListDeutsch.T_LanguagList[99]:='';
T_ErrorList.asErrorListDeutsch.T_LanguagList[100]:='';
T_ErrorList.asErrorListDeutsch.T_LanguagList[101]:='';
T_ErrorList.asErrorListDeutsch.T_LanguagList[102]:='';
T_ErrorList.asErrorListDeutsch.T_LanguagList[103]:='';
T_ErrorList.asErrorListDeutsch.T_LanguagList[104]:='';
T_ErrorList.asErrorListDeutsch.T_LanguagList[105]:='';
T_ErrorList.asErrorListDeutsch.T_LanguagList[106]:='';
T_ErrorList.asErrorListDeutsch.T_LanguagList[107]:='';
T_ErrorList.asErrorListDeutsch.T_LanguagList[108]:='';
T_ErrorList.asErrorListDeutsch.T_LanguagList[109]:='';
T_ErrorList.asErrorListDeutsch.T_LanguagList[110]:='';
T_ErrorList.asErrorListDeutsch.T_LanguagList[111]:='';
T_ErrorList.asErrorListDeutsch.T_LanguagList[112]:='';
T_ErrorList.asErrorListDeutsch.T_LanguagList[113]:='';
T_ErrorList.asErrorListDeutsch.T_LanguagList[114]:='';
T_ErrorList.asErrorListDeutsch.T_LanguagList[115]:='';
T_ErrorList.asErrorListDeutsch.T_LanguagList[116]:='';
T_ErrorList.asErrorListDeutsch.T_LanguagList[117]:='';
T_ErrorList.asErrorListDeutsch.T_LanguagList[118]:='';
T_ErrorList.asErrorListDeutsch.T_LanguagList[119]:='';
T_ErrorList.asErrorListDeutsch.T_LanguagList[120]:='';
T_ErrorList.asErrorListDeutsch.T_LanguagList[121]:='';
T_ErrorList.asErrorListDeutsch.T_LanguagList[122]:='';
T_ErrorList.asErrorListDeutsch.T_LanguagList[123]:='';
T_ErrorList.asErrorListDeutsch.T_LanguagList[124]:='';
T_ErrorList.asErrorListDeutsch.T_LanguagList[125]:='';
T_ErrorList.asErrorListDeutsch.T_LanguagList[126]:='';
T_ErrorList.asErrorListDeutsch.T_LanguagList[127]:='';
T_ErrorList.asErrorListDeutsch.T_LanguagList[128]:='';
T_ErrorList.asErrorListDeutsch.T_LanguagList[129]:='';
T_ErrorList.asErrorListDeutsch.T_LanguagList[130]:='';
T_ErrorList.asErrorListDeutsch.T_LanguagList[131]:='';
T_ErrorList.asErrorListDeutsch.T_LanguagList[132]:='';
T_ErrorList.asErrorListDeutsch.T_LanguagList[133]:='';
T_ErrorList.asErrorListDeutsch.T_LanguagList[134]:='';
T_ErrorList.asErrorListDeutsch.T_LanguagList[135]:='';
T_ErrorList.asErrorListDeutsch.T_LanguagList[136]:='';
T_ErrorList.asErrorListDeutsch.T_LanguagList[137]:='';
T_ErrorList.asErrorListDeutsch.T_LanguagList[138]:='';
T_ErrorList.asErrorListDeutsch.T_LanguagList[139]:='';
T_ErrorList.asErrorListDeutsch.T_LanguagList[140]:='';
T_ErrorList.asErrorListDeutsch.T_LanguagList[141]:='';
T_ErrorList.asErrorListDeutsch.T_LanguagList[142]:='';
T_ErrorList.asErrorListDeutsch.T_LanguagList[143]:='';
T_ErrorList.asErrorListDeutsch.T_LanguagList[144]:='';
T_ErrorList.asErrorListDeutsch.T_LanguagList[145]:='';
T_ErrorList.asErrorListDeutsch.T_LanguagList[146]:='';
T_ErrorList.asErrorListDeutsch.T_LanguagList[147]:='';
T_ErrorList.asErrorListDeutsch.T_LanguagList[148]:='';
T_ErrorList.asErrorListDeutsch.T_LanguagList[149]:='';
T_ErrorList.asErrorListDeutsch.T_LanguagList[150]:='';
T_ErrorList.asErrorListDeutsch.T_LanguagList[151]:='';
T_ErrorList.asErrorListDeutsch.T_LanguagList[152]:='';
T_ErrorList.asErrorListDeutsch.T_LanguagList[153]:='';
T_ErrorList.asErrorListDeutsch.T_LanguagList[154]:='';
T_ErrorList.asErrorListDeutsch.T_LanguagList[155]:='';
T_ErrorList.asErrorListDeutsch.T_LanguagList[156]:='';
T_ErrorList.asErrorListDeutsch.T_LanguagList[157]:='';
T_ErrorList.asErrorListDeutsch.T_LanguagList[158]:='';
T_ErrorList.asErrorListDeutsch.T_LanguagList[159]:='';
T_ErrorList.asErrorListDeutsch.T_LanguagList[160]:='';
T_ErrorList.asErrorListDeutsch.T_LanguagList[161]:='';
T_ErrorList.asErrorListDeutsch.T_LanguagList[162]:='';
T_ErrorList.asErrorListDeutsch.T_LanguagList[163]:='';
T_ErrorList.asErrorListDeutsch.T_LanguagList[164]:='';
T_ErrorList.asErrorListDeutsch.T_LanguagList[165]:='';
T_ErrorList.asErrorListDeutsch.T_LanguagList[166]:='';
T_ErrorList.asErrorListDeutsch.T_LanguagList[167]:='';
T_ErrorList.asErrorListDeutsch.T_LanguagList[168]:='';
T_ErrorList.asErrorListDeutsch.T_LanguagList[169]:='';
T_ErrorList.asErrorListDeutsch.T_LanguagList[170]:='';
T_ErrorList.asErrorListDeutsch.T_LanguagList[171]:='';
T_ErrorList.asErrorListDeutsch.T_LanguagList[172]:='';

(* Static Francais Error List *)
T_ErrorList.asErrorListFrancais.T_LanguagList[1]:='Internal problem, should never appear';
T_ErrorList.asErrorListFrancais.T_LanguagList[2]:='Antivalence error of the motor encoder';
T_ErrorList.asErrorListFrancais.T_LanguagList[3]:='Encoder counter error, >+/- 4 inc';
T_ErrorList.asErrorListFrancais.T_LanguagList[4]:='Mster encoder X7 counter error, >+/- 4 inc';
T_ErrorList.asErrorListFrancais.T_LanguagList[5]:='Heat sink temperature to high (>80°)';
T_ErrorList.asErrorListFrancais.T_LanguagList[6]:='Low voltage (<18V) of the +24V logic supply';
T_ErrorList.asErrorListFrancais.T_LanguagList[7]:='High voltage X10 (>180V) of the motor power supply';
T_ErrorList.asErrorListFrancais.T_LanguagList[8]:='Low voltage X10 (<24V) of the motor power supply';
T_ErrorList.asErrorListFrancais.T_LanguagList[9]:='Short circuit in the motor phase A';
T_ErrorList.asErrorListFrancais.T_LanguagList[10]:='Short circuit in the motor phase B';
T_ErrorList.asErrorListFrancais.T_LanguagList[11]:='Short circuit of a digital output';
T_ErrorList.asErrorListFrancais.T_LanguagList[12]:='Digital input ENABLE going to low level';
T_ErrorList.asErrorListFrancais.T_LanguagList[13]:='Exceed max. countouring error ';
T_ErrorList.asErrorListFrancais.T_LanguagList[14]:='Rotation speed to high, can not read encoder signal';
T_ErrorList.asErrorListFrancais.T_LanguagList[15]:='Can not find the commutation';
T_ErrorList.asErrorListFrancais.T_LanguagList[16]:='CAN-Communication broken by Node Guarding';
T_ErrorList.asErrorListFrancais.T_LanguagList[17]:='I^2t- Controlling triggered (current limit)';
T_ErrorList.asErrorListFrancais.T_LanguagList[18]:='ADS communication error';
T_ErrorList.asErrorListFrancais.T_LanguagList[19]:='Axis function time out error';
T_ErrorList.asErrorListFrancais.T_LanguagList[20]:='Axis function not implemented';
T_ErrorList.asErrorListFrancais.T_LanguagList[21]:='No HDD free resource, time out';
T_ErrorList.asErrorListFrancais.T_LanguagList[22]:='HDD error, no file found';
T_ErrorList.asErrorListFrancais.T_LanguagList[23]:='Axis Parameter File, wrong syntax';
T_ErrorList.asErrorListFrancais.T_LanguagList[24]:='Wrong Para Fct: Read Axis Parameter';
T_ErrorList.asErrorListFrancais.T_LanguagList[25]:='Limit End Switch Active';
T_ErrorList.asErrorListFrancais.T_LanguagList[26]:='PDOMapping Para File, wrong syntax';
T_ErrorList.asErrorListFrancais.T_LanguagList[27]:='Wrong Para Fct: Read PDOMapping Parameter';
T_ErrorList.asErrorListFrancais.T_LanguagList[28]:='No Axis Power Supply';
T_ErrorList.asErrorListFrancais.T_LanguagList[29]:='Wrong Para Fct: Move velocity';
T_ErrorList.asErrorListFrancais.T_LanguagList[30]:='Can not move, no power supply';
T_ErrorList.asErrorListFrancais.T_LanguagList[31]:='Wrong Para Fct: Move position absolute';
T_ErrorList.asErrorListFrancais.T_LanguagList[32]:='Wrong Para Fct: Move position relative';
T_ErrorList.asErrorListFrancais.T_LanguagList[33]:='Wrong Para Fct: Move referencing';
T_ErrorList.asErrorListFrancais.T_LanguagList[34]:='Fct CalcAnlgeRefIndex:Ref.Sensor not found';
T_ErrorList.asErrorListFrancais.T_LanguagList[35]:='Wrong Para Fct: Send Axis Parameter';
T_ErrorList.asErrorListFrancais.T_LanguagList[36]:='Wrong Para Fct: Send PDOMapping Parameter';
T_ErrorList.asErrorListFrancais.T_LanguagList[37]:='Wrong Para Fct: Master/Slave';
T_ErrorList.asErrorListFrancais.T_LanguagList[38]:='Axis general error';
T_ErrorList.asErrorListFrancais.T_LanguagList[39]:='ToolLeft: Wrong configuration or Axis missing';
T_ErrorList.asErrorListFrancais.T_LanguagList[40]:='ToolCenter: Wrong configuration or Axis missing';
T_ErrorList.asErrorListFrancais.T_LanguagList[41]:='ToolRight: Wrong configuration or Axis missing';
T_ErrorList.asErrorListFrancais.T_LanguagList[42]:='ToolFeeder: Wrong configuration or Axis missing';
T_ErrorList.asErrorListFrancais.T_LanguagList[43]:='GrindFeeder: Wrong configuration or Axis missing';
T_ErrorList.asErrorListFrancais.T_LanguagList[44]:='BoxId general error';
T_ErrorList.asErrorListFrancais.T_LanguagList[45]:='Cyl. Function not implemented';
T_ErrorList.asErrorListFrancais.T_LanguagList[46]:='Sensor down not active';
T_ErrorList.asErrorListFrancais.T_LanguagList[47]:='Sensor up not active';
T_ErrorList.asErrorListFrancais.T_LanguagList[48]:='Cyl. general error';
T_ErrorList.asErrorListFrancais.T_LanguagList[49]:='File for profile not found';
T_ErrorList.asErrorListFrancais.T_LanguagList[50]:='Profile file not found: ';
T_ErrorList.asErrorListFrancais.T_LanguagList[51]:='--> Load static default parameter';
T_ErrorList.asErrorListFrancais.T_LanguagList[52]:='Machine is not referenced';
T_ErrorList.asErrorListFrancais.T_LanguagList[53]:='Settled parameter for ToolLength is to long';
T_ErrorList.asErrorListFrancais.T_LanguagList[54]:='Settled parameter for ToolLength is to short';
T_ErrorList.asErrorListFrancais.T_LanguagList[55]:='Settled parameter for ToolDiameter is to big';
T_ErrorList.asErrorListFrancais.T_LanguagList[56]:='Settled parameter for ToolDiameter is to small';
T_ErrorList.asErrorListFrancais.T_LanguagList[57]:='Tool is not clamped';
T_ErrorList.asErrorListFrancais.T_LanguagList[58]:='ToolTension is not active';
T_ErrorList.asErrorListFrancais.T_LanguagList[59]:='ToolFeeeder is not on the StartPosition';
T_ErrorList.asErrorListFrancais.T_LanguagList[60]:='At least one Axis is busy';
T_ErrorList.asErrorListFrancais.T_LanguagList[61]:='Undefined Station error';
T_ErrorList.asErrorListFrancais.T_LanguagList[62]:='At least a passage of a section is not equal';
T_ErrorList.asErrorListFrancais.T_LanguagList[63]:='On the MicroWire it is not possible to Referencing';
T_ErrorList.asErrorListFrancais.T_LanguagList[64]:='Undefined Machine Error';
T_ErrorList.asErrorListFrancais.T_LanguagList[65]:='At least one Ecostep CANOpen Controller failed!';
T_ErrorList.asErrorListFrancais.T_LanguagList[66]:='No Air Pressure';
T_ErrorList.asErrorListFrancais.T_LanguagList[67]:='At least one settled diameter is bigger than ToolDiameter';
T_ErrorList.asErrorListFrancais.T_LanguagList[68]:='ToolTension is active';
T_ErrorList.asErrorListFrancais.T_LanguagList[69]:='';
T_ErrorList.asErrorListFrancais.T_LanguagList[70]:='';
T_ErrorList.asErrorListFrancais.T_LanguagList[71]:='';
T_ErrorList.asErrorListFrancais.T_LanguagList[72]:='';
T_ErrorList.asErrorListFrancais.T_LanguagList[73]:='';
T_ErrorList.asErrorListFrancais.T_LanguagList[74]:='';
T_ErrorList.asErrorListFrancais.T_LanguagList[75]:='';
T_ErrorList.asErrorListFrancais.T_LanguagList[76]:='';
T_ErrorList.asErrorListFrancais.T_LanguagList[77]:='';
T_ErrorList.asErrorListFrancais.T_LanguagList[78]:='';
T_ErrorList.asErrorListFrancais.T_LanguagList[79]:='';
T_ErrorList.asErrorListFrancais.T_LanguagList[80]:='';
T_ErrorList.asErrorListFrancais.T_LanguagList[81]:='';
T_ErrorList.asErrorListFrancais.T_LanguagList[82]:='';
T_ErrorList.asErrorListFrancais.T_LanguagList[83]:='';
T_ErrorList.asErrorListFrancais.T_LanguagList[84]:='';
T_ErrorList.asErrorListFrancais.T_LanguagList[85]:='';
T_ErrorList.asErrorListFrancais.T_LanguagList[86]:='';
T_ErrorList.asErrorListFrancais.T_LanguagList[87]:='';
T_ErrorList.asErrorListFrancais.T_LanguagList[88]:='';
T_ErrorList.asErrorListFrancais.T_LanguagList[89]:='';
T_ErrorList.asErrorListFrancais.T_LanguagList[90]:='';
T_ErrorList.asErrorListFrancais.T_LanguagList[91]:='';
T_ErrorList.asErrorListFrancais.T_LanguagList[92]:='';
T_ErrorList.asErrorListFrancais.T_LanguagList[93]:='';
T_ErrorList.asErrorListFrancais.T_LanguagList[94]:='';
T_ErrorList.asErrorListFrancais.T_LanguagList[95]:='';
T_ErrorList.asErrorListFrancais.T_LanguagList[96]:='';
T_ErrorList.asErrorListFrancais.T_LanguagList[97]:='';
T_ErrorList.asErrorListFrancais.T_LanguagList[98]:='';
T_ErrorList.asErrorListFrancais.T_LanguagList[99]:='';
T_ErrorList.asErrorListFrancais.T_LanguagList[100]:='';
T_ErrorList.asErrorListFrancais.T_LanguagList[101]:='';
T_ErrorList.asErrorListFrancais.T_LanguagList[102]:='';
T_ErrorList.asErrorListFrancais.T_LanguagList[103]:='';
T_ErrorList.asErrorListFrancais.T_LanguagList[104]:='';
T_ErrorList.asErrorListFrancais.T_LanguagList[105]:='';
T_ErrorList.asErrorListFrancais.T_LanguagList[106]:='';
T_ErrorList.asErrorListFrancais.T_LanguagList[107]:='';
T_ErrorList.asErrorListFrancais.T_LanguagList[108]:='';
T_ErrorList.asErrorListFrancais.T_LanguagList[109]:='';
T_ErrorList.asErrorListFrancais.T_LanguagList[110]:='';
T_ErrorList.asErrorListFrancais.T_LanguagList[111]:='';
T_ErrorList.asErrorListFrancais.T_LanguagList[112]:='';
T_ErrorList.asErrorListFrancais.T_LanguagList[113]:='';
T_ErrorList.asErrorListFrancais.T_LanguagList[114]:='';
T_ErrorList.asErrorListFrancais.T_LanguagList[115]:='';
T_ErrorList.asErrorListFrancais.T_LanguagList[116]:='';
T_ErrorList.asErrorListFrancais.T_LanguagList[117]:='';
T_ErrorList.asErrorListFrancais.T_LanguagList[118]:='';
T_ErrorList.asErrorListFrancais.T_LanguagList[119]:='';
T_ErrorList.asErrorListFrancais.T_LanguagList[120]:='';
T_ErrorList.asErrorListFrancais.T_LanguagList[121]:='';
T_ErrorList.asErrorListFrancais.T_LanguagList[122]:='';
T_ErrorList.asErrorListFrancais.T_LanguagList[123]:='';
T_ErrorList.asErrorListFrancais.T_LanguagList[124]:='';
T_ErrorList.asErrorListFrancais.T_LanguagList[125]:='';
T_ErrorList.asErrorListFrancais.T_LanguagList[126]:='';
T_ErrorList.asErrorListFrancais.T_LanguagList[127]:='';
T_ErrorList.asErrorListFrancais.T_LanguagList[128]:='';
T_ErrorList.asErrorListFrancais.T_LanguagList[129]:='';
T_ErrorList.asErrorListFrancais.T_LanguagList[130]:='';
T_ErrorList.asErrorListFrancais.T_LanguagList[131]:='';
T_ErrorList.asErrorListFrancais.T_LanguagList[132]:='';
T_ErrorList.asErrorListFrancais.T_LanguagList[133]:='';
T_ErrorList.asErrorListFrancais.T_LanguagList[134]:='';
T_ErrorList.asErrorListFrancais.T_LanguagList[135]:='';
T_ErrorList.asErrorListFrancais.T_LanguagList[136]:='';
T_ErrorList.asErrorListFrancais.T_LanguagList[137]:='';
T_ErrorList.asErrorListFrancais.T_LanguagList[138]:='';
T_ErrorList.asErrorListFrancais.T_LanguagList[139]:='';
T_ErrorList.asErrorListFrancais.T_LanguagList[140]:='';
T_ErrorList.asErrorListFrancais.T_LanguagList[141]:='';
T_ErrorList.asErrorListFrancais.T_LanguagList[142]:='';
T_ErrorList.asErrorListFrancais.T_LanguagList[143]:='';
T_ErrorList.asErrorListFrancais.T_LanguagList[144]:='';
T_ErrorList.asErrorListFrancais.T_LanguagList[145]:='';
T_ErrorList.asErrorListFrancais.T_LanguagList[146]:='';
T_ErrorList.asErrorListFrancais.T_LanguagList[147]:='';
T_ErrorList.asErrorListFrancais.T_LanguagList[148]:='';
T_ErrorList.asErrorListFrancais.T_LanguagList[149]:='';
T_ErrorList.asErrorListFrancais.T_LanguagList[150]:='';
T_ErrorList.asErrorListFrancais.T_LanguagList[151]:='';
T_ErrorList.asErrorListFrancais.T_LanguagList[152]:='';
T_ErrorList.asErrorListFrancais.T_LanguagList[153]:='';
T_ErrorList.asErrorListFrancais.T_LanguagList[154]:='';
T_ErrorList.asErrorListFrancais.T_LanguagList[155]:='';
T_ErrorList.asErrorListFrancais.T_LanguagList[156]:='';
T_ErrorList.asErrorListFrancais.T_LanguagList[157]:='';
T_ErrorList.asErrorListFrancais.T_LanguagList[158]:='';
T_ErrorList.asErrorListFrancais.T_LanguagList[159]:='';
T_ErrorList.asErrorListFrancais.T_LanguagList[160]:='';
T_ErrorList.asErrorListFrancais.T_LanguagList[161]:='';
T_ErrorList.asErrorListFrancais.T_LanguagList[162]:='';
T_ErrorList.asErrorListFrancais.T_LanguagList[163]:='';
T_ErrorList.asErrorListFrancais.T_LanguagList[164]:='';
T_ErrorList.asErrorListFrancais.T_LanguagList[165]:='';
T_ErrorList.asErrorListFrancais.T_LanguagList[166]:='';
T_ErrorList.asErrorListFrancais.T_LanguagList[167]:='';
T_ErrorList.asErrorListFrancais.T_LanguagList[168]:='';
T_ErrorList.asErrorListFrancais.T_LanguagList[169]:='';
T_ErrorList.asErrorListFrancais.T_LanguagList[170]:='';
T_ErrorList.asErrorListFrancais.T_LanguagList[171]:='';
T_ErrorList.asErrorListFrancais.T_LanguagList[172]:='';
END_FUNCTION_BLOCK

(* POU GENERAL/FB_BIOSPARAMETER, ST *)
FUNCTION_BLOCK FB_BIOSPARAMETER
VAR_INPUT
	dwBIOSPasswordPage:DWORD;		(* Page number of the BIOS password page *)
	dwBIOSParameterPage:DWORD;		(* Page number of the BIOS parameter page *)
	T_TwinSafeOut:ST_TWINSAFE_OUT;	(* Output of the TwinSAFE components *)
END_VAR
VAR_IN_OUT
	T_Visu:ST_QVIS;						(* Data structure of the visualisation *)
	T_HDD:ST_HDD;						(* Data structure of the File Management *)
	T_NovRam : ST_NOVRAM;				(* Data structure of the NovRam *)
	T_CtrlePanel:ST_CTRLEPANEL;		(* Data structure of the ControlPanel *)
	T_DeviceID:ST_DEVICEID;				(* Data structure of the Device components *)
	T_BoxID:ST_BOXID;					(* Data structure of the components with the BoxId *)
	T_Profile:ST_PROFILE;				(* Data structure of the Profile management *)
END_VAR
VAR_OUTPUT
END_VAR
VAR
	TONShowMessage: TON;
	xChangeToBIOSPassword: BOOL;
	xChangeToBIOSParameter: BOOL;
	xSaveBIOSParameterToNovRAM: BOOL;
	xCopyBIOSParameter: BOOL;
	xReadFirstTimeParameter: BOOL;
	iStepSaveToNovRAM: INT;
	iStepReadFirstTimeParameter: INT;
	xCheckMsgBoxActive: BOOL;
(* Random *)
	fbGetCpuAccount:GETCPUCOUNTER;
	fbPwSystem:FBPW_SYSTEM;
	iPwSystem:INT;
	xNovRAMParaReaded: BOOL;
	xTmp: BOOL;
END_VAR
(****************************************************************************************************************************************************)
(***********     This Functionblock gives the possibility to set the bios parameter, with input a SystemLevel password     ************)
(****************************************************************************************************************************************************)
(* Managing BIOS Parameter on Startup *)
	IF (T_Visu.ptrT_ExchgParam^.T_Visu.T_Message.iStateBIOS <> 0) THEN
		TONShowMessage(IN:=TRUE,PT:=T#3s);
		IF TONShowMessage.Q THEN
			T_Visu.ptrT_ExchgParam^.T_Visu.T_Message.iStateBIOS:=0;
		END_IF;
	ELSE
		TONShowMessage(IN:=FALSE);
	END_IF;
	xCheckMsgBoxActive:=	(T_Visu.ptrT_ExchgParam^.T_SafetyCtrl.bStateMessageError <> 0) OR
							(T_Visu.ptrT_ExchgParam^.T_SafetyCtrl.bStateMessageInfo <> 0) OR
							(T_Visu.ptrT_ExchgParam^.T_SafetyCtrl.bStateMessageWarning <> 0);
	IF ((T_Visu.T_PlcParam.dwActualPage = 0) AND NOT(T_Visu.T_CtrleVisu.xExecute) AND T_Visu.T_CtrleVisu.xDone) OR xCheckMsgBoxActive THEN
		xChangeToBIOSPassword:=FALSE;
		xChangeToBIOSParameter:=FALSE;
		xSaveBIOSParameterToNovRAM:=FALSE;
		xCopyBIOSParameter:=FALSE;
		xReadFirstTimeParameter:=FALSE;
		iStepSaveToNovRAM:=1;
		iStepReadFirstTimeParameter:=1;
		T_Visu.ptrT_ExchgParam^.T_Visu.T_Message.iStateBIOS:=0;
		IF (T_Visu.ptrT_ExchgParam^.T_Config.iEditParam = DWORD_TO_INT(dwBIOSParameterPage)) THEN
			T_Visu.ptrT_ExchgParam^.T_Config.iEditParam:=0;
		END_IF;
	END_IF;
	IF (T_Visu.T_PlcParam.dwActualPage = dwBIOSPasswordPage) OR (T_Visu.T_PlcParam.dwActualPage = dwBIOSParameterPage) THEN
		IF (T_Visu.ptrT_ExchgParam^.T_SafetyCtrl.iStateStartPage = 2) THEN	(* check if external relase button has been pressed *)
			IF NOT(T_Visu.T_CtrleVisu.xExecute) AND T_Visu.T_CtrleVisu.xDone THEN
				T_Visu.T_PlcParam.dwSetNewPage:=0;
				T_Visu.T_CtrleVisu.iFunction:=1;
				T_Visu.T_CtrleVisu.xExecute:=TRUE;
			END_IF;
		END_IF;
	END_IF;
	(* check if the function button F1 is pressed-->if it is pressed the change to the BIOS password page *)
	IF NOT(xChangeToBIOSPassword) THEN
		IF (T_Visu.T_PlcParam.dwActualPage = 0) AND NOT(T_StartUp.T_State.xCompleted) THEN
			IF (T_Visu.ptrT_ExchgParam^.T_SafetyCtrl.iStateStartPage = 1) AND NOT(T_TwinSafeOut.QxContactor_K3) AND NOT(T_TwinSafeOut.QxContactor_K4) THEN
				IF T_Visu.ptrT_ExchgParam^.T_BtFunctionPanel.wActivBt = 16#1 THEN
					T_Visu.ptrT_ExchgParam^.T_BtFunctionPanel.wActivBt:=0;
					IF NOT(T_Visu.T_CtrleVisu.xExecute) AND T_Visu.T_CtrleVisu.xDone THEN
						T_Visu.ptrT_ExchgParam^.T_Visu.T_Message.iStateBIOS:=0;
						xChangeToBIOSPassword:=TRUE;
						T_Visu.T_PlcParam.dwSetNewPage:=dwBIOSPasswordPage;
						T_Visu.T_CtrleVisu.iFunction:=1;
						T_Visu.T_CtrleVisu.xExecute:=TRUE;
						fbGetCpuAccount;
						fbPwSystem(	dwCounter:=fbGetCpuAccount.fbGetCpuCounter.dwCpuCntHi+fbGetCpuAccount.fbGetCpuCounter.dwCpuCntLo,
									iRandom=>T_Visu.ptrT_ExchgParam^.T_Visu.T_Level.iRandom,
									iPwSystem=>iPwSystem);
					END_IF;
				END_IF;
			END_IF;
		END_IF;
	END_IF;
	(* check the settled password *)
	IF xChangeToBIOSPassword THEN
		IF (T_Visu.T_PlcParam.dwActualPage = dwBIOSPasswordPage) THEN
			IF T_Visu.ptrT_ExchgParam^.T_Visu.xKey_Escape THEN	(* ESC Button for exit and go to the Startpage *)
				T_Visu.ptrT_ExchgParam^.T_Visu.xKey_Escape:=FALSE;
				IF NOT(T_Visu.T_CtrleVisu.xExecute) AND T_Visu.T_CtrleVisu.xDone THEN
					xChangeToBIOSPassword:=FALSE;
					T_Visu.T_PlcParam.dwSetNewPage:=0;
					T_Visu.T_CtrleVisu.iFunction:=1;
					T_Visu.T_CtrleVisu.xExecute:=TRUE;
					T_Visu.ptrT_ExchgParam^.T_Visu.T_Level.iPwSystem:=999;
				END_IF;
			END_IF;
			IF (T_Visu.ptrT_ExchgParam^.T_Visu.T_Level.iPwSystem = iPwSystem) THEN
				T_Visu.ptrT_ExchgParam^.T_Visu.T_Message.iStateBIOS:=0;
				T_Visu.ptrT_ExchgParam^.T_Visu.T_Level.iPwSystem:=999;
				IF NOT(T_Visu.T_CtrleVisu.xExecute) AND T_Visu.T_CtrleVisu.xDone THEN
					xChangeToBIOSPassword:=FALSE;
					xChangeToBIOSParameter:=TRUE;
					T_Visu.T_PlcParam.dwSetNewPage:=dwBIOSParameterPage;
					T_Visu.T_CtrleVisu.iFunction:=1;
					T_Visu.T_CtrleVisu.xExecute:=TRUE;
					IF NOT(T_NovRam.T_Ctrle.xFirstRead) THEN
						xReadFirstTimeParameter:=TRUE;
					ELSE
						xCopyBIOSParameter:=TRUE;
					END_IF;
				END_IF;
			END_IF;
			IF (T_Visu.ptrT_ExchgParam^.T_Visu.T_Level.iPwSystem <> 999) THEN
				IF (T_Visu.ptrT_ExchgParam^.T_Visu.T_Level.iPwSystem <> iPwSystem) THEN
					T_Visu.ptrT_ExchgParam^.T_Visu.T_Message.iStateBIOS:=2;	(* Wrong password *)
					T_Visu.ptrT_ExchgParam^.T_Visu.T_Level.iPwSystem:=999;
				END_IF;
			END_IF;
		END_IF;
	END_IF;
	(* the edit parameterlist is now active *)
	IF xChangeToBIOSParameter AND NOT(xReadFirstTimeParameter) THEN
		T_Visu.ptrT_ExchgParam^.T_Config.iEditParam:=DWORD_TO_INT(dwBIOSParameterPage);
		IF (T_Visu.T_PlcParam.dwActualPage = dwBIOSParameterPage) AND NOT(xReadFirstTimeParameter) AND NOT(xSaveBIOSParameterToNovRAM) AND NOT(xCopyBIOSParameter) THEN
			IF T_Visu.ptrT_ExchgParam^.T_Visu.xKey_Escape THEN	(* ESC Button for exit and go to the Startpage *)
				T_Visu.ptrT_ExchgParam^.T_Visu.xKey_Escape:=FALSE;
				IF NOT(T_Visu.T_CtrleVisu.xExecute) AND T_Visu.T_CtrleVisu.xDone THEN
					xChangeToBIOSParameter:=FALSE;
					xSaveBIOSParameterToNovRAM:=FALSE;
					xCopyBIOSParameter:=TRUE;
					T_Visu.T_PlcParam.dwSetNewPage:=0;
					T_Visu.T_CtrleVisu.iFunction:=1;
					T_Visu.T_CtrleVisu.xExecute:=TRUE;
				END_IF;
			END_IF;
			IF (UDINT_TO_WORD(T_CtrlePanel.udiButton) = 16#200) AND NOT(xSaveBIOSParameterToNovRAM) THEN	(* Right Panel Button for save Parameter *)
				T_Visu.ptrT_ExchgParam^.T_Visu.T_Message.iStateBIOS:=1;	(* Parameter saved *)
				xSaveBIOSParameterToNovRAM:=TRUE;
				xCopyBIOSParameter:=FALSE;
				iStepSaveToNovRAM:=1;
			END_IF;
		END_IF;
	END_IF;
	(* save the settled parameter to the NovRam *)
	IF xSaveBIOSParameterToNovRAM THEN
		CASE iStepSaveToNovRAM OF
		1:	IF xNovRAMParaReaded THEN
				(* 30.11.2010 KFS: {	*)
				IF ( T_NovRam.T_Data.T_Standard.T_MachineConfig.rConfigMaxToolLength <> T_Visu.ptrT_ExchgParam^.T_StationCommon.rConfigMaxToolLength) THEN
					T_NovRam.T_Data.T_Standard.T_MachineConfig.rConfigMaxToolLengthOriginal:=0.0;
				END_IF;
				(* 30.11.2010 KFS:	}	*)
				T_NovRam.T_Data.T_Standard.T_MachineConfig.iConfigMachineType:=T_Visu.ptrT_ExchgParam^.T_StationCommon.iConfigMachineType;
				T_NovRam.T_Data.T_Standard.T_MachineConfig.iConfigAxisType:=T_Visu.ptrT_ExchgParam^.T_StationCommon.iConfigAxisType;
				T_NovRam.T_Data.T_Standard.T_MachineConfig.iConfigVisuNavigation:=T_Visu.ptrT_ExchgParam^.T_StationCommon.iConfigVisuNavigation;
				T_NovRam.T_Data.T_Standard.T_MachineConfig.rConfigMaxToolLength:=T_Visu.ptrT_ExchgParam^.T_StationCommon.rConfigMaxToolLength;
				T_NovRAM.T_Ctrle.iFunction:=2;
				T_NovRAM.T_Ctrle.xExecute:=TRUE;
				iStepSaveToNovRAM:=10;
			ELSE
				iStepSaveToNovRAM:=1;
				xSaveBIOSParameterToNovRAM:=FALSE;
			END_IF;
		10:	IF NOT(T_NovRAM.T_Ctrle.xExecute) AND T_NovRAM.T_Ctrle.xDone THEN
				iStepSaveToNovRAM:=1;
				xSaveBIOSParameterToNovRAM:=FALSE;
				T_Visu.T_CtrleVisu.xReset:=TRUE;	(* Exit the BIOS Parameter Page *)
			END_IF;
		END_CASE;
	END_IF;
	(* copy the NovRam config parameter to the visu structure *)
	IF xCopyBIOSParameter THEN
		IF xNovRAMParaReaded THEN
			T_Visu.ptrT_ExchgParam^.T_StationCommon.iConfigMachineType:=T_NovRam.T_Data.T_Standard.T_MachineConfig.iConfigMachineType;
			T_Visu.ptrT_ExchgParam^.T_StationCommon.iConfigAxisType:=T_NovRam.T_Data.T_Standard.T_MachineConfig.iConfigAxisType;
			T_Visu.ptrT_ExchgParam^.T_StationCommon.iConfigVisuNavigation:=T_NovRam.T_Data.T_Standard.T_MachineConfig.iConfigVisuNavigation;
			T_Visu.ptrT_ExchgParam^.T_StationCommon.rConfigMaxToolLength:=T_NovRam.T_Data.T_Standard.T_MachineConfig.rConfigMaxToolLength;
			T_Visu.ptrT_ExchgParam^.T_StationCommon.rConfigMaxToolLengthOriginal:=T_NovRam.T_Data.T_Standard.T_MachineConfig.rConfigMaxToolLengthOriginal;
			xCopyBIOSParameter:=FALSE;
		ELSE
			xCopyBIOSParameter:=FALSE;
		END_IF;
	END_IF;
	(* Init the Hardware for read the first time the parameter *)
	IF xReadFirstTimeParameter THEN
		CASE iStepReadFirstTimeParameter OF
		1:	T_HDD.T_Ctrle.xReset:=TRUE;
			T_DeviceID.T_Ctrle.xReset:=TRUE;
			T_BoxID.T_Ctrle.xReset:=TRUE;
			T_NovRAM.T_Ctrle.xReset:=TRUE;
			T_Profile.T_Ctrle.xReset:=TRUE;
			(* next step *)
			iStepReadFirstTimeParameter:=10;
			(* waiting reset confirmation *)
		10:	xTmp:=	T_HDD.T_Ctrle.xDone
					AND T_DeviceID.T_Ctrle.xDone
					AND T_NovRAM.T_Ctrle.xDone
					AND T_BoxID.T_Ctrle.xDone
					AND T_Profile.T_Ctrle.xDone;
			IF xTmp THEN  iStepReadFirstTimeParameter:=20; END_IF
		20:	(* PLC name *)
			T_DeviceID.T_CX1020.sDeviceName:='CX1000_PLC';
			(* feldbus name *)
			T_DeviceID.T_CANOpenMaster.sDeviceName:='CANOpenMaster';
			T_DeviceID.T_CANOpenMaster.xDeviceOption:=TRUE;
			T_DeviceID.T_LightbusMaster.sDeviceName:='LightbusMaster';
			T_DeviceID.T_LightbusMaster.xDeviceOption:=TRUE;
			(* NovRAM *)
			T_DeviceID.T_NovRAM.sDeviceName:='NovRAM';
			(* read device ID *)
			T_DeviceID.T_Ctrle.xExecute:=TRUE;
			(* next step *)
			iStepReadFirstTimeParameter:=30;
		(* waiting ID confirmation, Start BoxID *)
		30:	IF NOT(T_DeviceID.T_Ctrle.xExecute) AND T_DeviceID.T_Ctrle.xDone THEN iStepReadFirstTimeParameter:=40; END_IF
		(* waiting Box ID confirmation *)
		40:	IF NOT(T_BoxID.T_Ctrle.xExecute) AND T_BoxID.T_Ctrle.xDone THEN
				(* next step *)
				iStepReadFirstTimeParameter:=50;
			END_IF
		50:	T_NovRAM.T_Ctrle.iFunction:=1;
			T_NovRam.T_Ctrle.xBlockReadFirstTime:=TRUE;
			T_NovRAM.T_Ctrle.xExecute:=TRUE;
			iStepReadFirstTimeParameter:=60;
		60:	IF NOT(T_NovRAM.T_Ctrle.xExecute) AND T_NovRAM.T_Ctrle.xDone THEN
				xNovRAMParaReaded:=TRUE;
				T_Visu.ptrT_ExchgParam^.T_StationCommon.iConfigMachineType:=T_NovRam.T_Data.T_Standard.T_MachineConfig.iConfigMachineType;
				T_Visu.ptrT_ExchgParam^.T_StationCommon.iConfigAxisType:=T_NovRam.T_Data.T_Standard.T_MachineConfig.iConfigAxisType;
				T_Visu.ptrT_ExchgParam^.T_StationCommon.iConfigVisuNavigation:=T_NovRam.T_Data.T_Standard.T_MachineConfig.iConfigVisuNavigation;
				T_Visu.ptrT_ExchgParam^.T_StationCommon.rConfigMaxToolLength:=T_NovRam.T_Data.T_Standard.T_MachineConfig.rConfigMaxToolLength;
				T_Visu.ptrT_ExchgParam^.T_StationCommon.rConfigMaxToolLengthOriginal:=T_NovRam.T_Data.T_Standard.T_MachineConfig.rConfigMaxToolLengthOriginal;
				xReadFirstTimeParameter:=FALSE;
				iStepReadFirstTimeParameter:=1;
			END_IF;
		END_CASE;
	END_IF;
END_FUNCTION_BLOCK

(* POU PRG_VISU_LAYER5/FB_VISU/FBPW_SYSTEM, ST *)
FUNCTION_BLOCK FBPW_SYSTEM
VAR_INPUT
	dwCounter:DWORD;		(* number for generate the key *)
END_VAR
VAR_OUTPUT
	iRandom:INT;				(* generated key number for the password *)
	iPwSystem:INT;			(* level of the password *)
END_VAR
VAR
	i:INT;
	iCounter:INT;
	sTmp:STRING;
END_VAR
(****************************************************************************************************************************************************)
(***********                           This Functionblock is for the dynamic password, it generate a key number                                     ************)
(****************************************************************************************************************************************************)
(*
	dynamic System password
	ex : Counter=12345 => pw=55
	formul : 1+2+3+4+5 + 40 = 55
*)

(* Init. value *)
	iPwSystem:=0;
(* Convert value *)
	iCounter:=DWORD_TO_INT(dwCounter);
	IF iCounter<0 THEN iCounter:=iCounter*-1; END_IF
(* Set Random value *)
	iRandom:=iCounter;
	sTmp:=INT_TO_STRING(iCounter);
(* Set System pw *)
	FOR i:=0 TO LEN(sTmp)-1 DO
		iPwSystem:=iPwSystem+STRING_TO_INT(MID(sTmp,1,LEN(sTmp)-i));
		IF i=1 THEN iPwSystem:=iPwSystem+STRING_TO_INT(MID(sTmp,1,LEN(sTmp)-i))*10; END_IF
	END_FOR
END_FUNCTION_BLOCK

(* POU PRG_PROCESS_LAYER4/FB_PROCESS/FB_ErrorMessage, ST *)
FUNCTION_BLOCK FB_ErrorMessage
VAR_INPUT
	diErrorNr : DINT;				(* input of the error number *)
	T_ErrorList:ST_ERROR_LIST;	(* data structure of the errolist *)
END_VAR
VAR_OUTPUT
	sErrorTextEnglish : STRING(100);	(* give the error text in english *)
	sErrorTextDeutsch : STRING(100);	(* give the error text in german *)
	sErrorTextFrancais : STRING(100);	(* give the error text in french *)
END_VAR
VAR
	sTmpText1:STRING(100);
	sTmpText2:STRING(100);
	diTmpErrorNr:DINT;
	ptrErrorList: POINTER TO ST_LANGUAGE_LIST;
	iCounterLanguage: INT;
	sTmpErrorText : STRING(100);
	diTmpDeletePrefix: DINT;
END_VAR
(****************************************************************************************************************************************************)
(***********                     This Functionblock calculate all errors of the machine an set the follow errornumber                         ************)
(****************************************************************************************************************************************************)
ptrErrorList:=ADR(T_ErrorList.asErrorListEnglish);	(* pointer of the errorlist, default english *)
sErrorTextEnglish:='';
sErrorTextDeutsch:='';
sErrorTextFrancais:='';
sTmpText1:='';
diTmpErrorNr:=0;
diTmpDeletePrefix:=0;
(* detect the error of the hardware, station or process *)
IF (diErrorNr >= 1000000) AND (diErrorNr < 2000000) THEN
	diTmpDeletePrefix:=1000000;
	sTmpText1:='ToolLeft: ';
END_IF;
IF (diErrorNr >= 2000000) AND (diErrorNr < 3000000) THEN
	diTmpDeletePrefix:=2000000;
	sTmpText1:='ToolCenter: ';
END_IF;
IF (diErrorNr >= 3000000) AND (diErrorNr < 4000000) THEN
	diTmpDeletePrefix:=3000000;
	sTmpText1:='ToolRight: ';
END_IF;
IF (diErrorNr >= 4000000) AND (diErrorNr < 5000000) THEN
	diTmpDeletePrefix:=4000000;
	sTmpText1:='ToolFeeder: ';
END_IF;
IF (diErrorNr >= 5000000) AND (diErrorNr < 6000000) THEN
	diTmpDeletePrefix:=5000000;
	sTmpText1:='GrindFeeder: ';
END_IF;
IF (diErrorNr >= 6000000) AND (diErrorNr < 7000000) THEN
	diTmpDeletePrefix:=6000000;
	sTmpText1:='ToolTension: ';
END_IF;
IF (diErrorNr >= 7000000) AND (diErrorNr < 8000000) THEN
	diTmpDeletePrefix:=7000000;
	sTmpText1:='BoxId Err: ';
END_IF;
IF (diErrorNr >= 8000000) AND (diErrorNr < 9000000) THEN
	diTmpDeletePrefix:=8000000;
	sTmpText1:='Station Err: ';
END_IF;

FOR iCounterLanguage:=1 TO 3 DO
	sTmpText2:='';
	sTmpErrorText:='';
	(* set the pointer for the errorlist of the language english, german or french *)
	IF (iCounterLanguage = 1) THEN	ptrErrorList:=ADR(T_ErrorList.asErrorListEnglish); END_IF;
	IF (iCounterLanguage = 2) THEN	ptrErrorList:=ADR(T_ErrorList.asErrorListDeutsch); END_IF;
	IF (iCounterLanguage = 3) THEN	ptrErrorList:=ADR(T_ErrorList.asErrorListFrancais); END_IF;
	IF (diErrorNr >= 0) AND (diErrorNr < 1000000) THEN
		CASE diErrorNr OF
			1:			sTmpText2:=ptrErrorList^.T_LanguagList[52];		(* 'Machine is not referenced' *)
			2:			sTmpText2:=ptrErrorList^.T_LanguagList[57];		(* 'Tool is not clamped' *)
			3:			sTmpText2:=ptrErrorList^.T_LanguagList[58];		(* 'ToolTension is not active' *)
			4:			sTmpText2:=ptrErrorList^.T_LanguagList[59];		(* 'ToolFeeeder is not on the StartPosition' *)
			5:			sTmpText2:=ptrErrorList^.T_LanguagList[63];		(* 'On the MicroWire it is not possible to Referencing' *)
			6:			sTmpText2:=ptrErrorList^.T_LanguagList[65];		(* 'At least one Ecostep CANOpen Controller failed!' *)
			7:			sTmpText2:=ptrErrorList^.T_LanguagList[66];		(* 'No Air Pressure' *)
			16#F201:		sTmpText2:=ptrErrorList^.T_LanguagList[53];		(* 'Settled parameter for ToolLength is to long' *)
			16#F202:		sTmpText2:=ptrErrorList^.T_LanguagList[54];		(* 'Settled parameter for ToolLength is to short' *)
			16#F203:		sTmpText2:=ptrErrorList^.T_LanguagList[55];		(* 'Settled parameter for ToolDiameter is to big' *)
			16#F204:		sTmpText2:=ptrErrorList^.T_LanguagList[56];		(* 'Settled parameter for ToolDiameter is to small' *)
			16#F205:		sTmpText2:=ptrErrorList^.T_LanguagList[62];		(* 'At least a passage of a section is not equal' *)
			16#F206:		sTmpText2:=ptrErrorList^.T_LanguagList[67];		(* 'At least one settled diameter is bigger than ToolDiameter' *)
		ELSE
						sTmpText2:=ptrErrorList^.T_LanguagList[64];		(* 'Undefined Machine Error' *)
		END_CASE;
		sTmpErrorText:=CONCAT(sTmpText1,sTmpText2);
		IF (iCounterLanguage = 1) THEN sErrorTextEnglish:=sTmpErrorText;	END_IF;
		IF (iCounterLanguage = 2) THEN sErrorTextDeutsch:=sTmpErrorText;	END_IF;
		IF (iCounterLanguage = 3) THEN sErrorTextFrancais:=sTmpErrorText;	END_IF;
	ELSE
		IF (diErrorNr >= 1000000) AND (diErrorNr < 6000000) THEN
			diTmpErrorNr:=diErrorNr - diTmpDeletePrefix;
			CASE diTmpErrorNr OF
			16#F201:		sTmpText2:=ptrErrorList^.T_LanguagList[20];	(* 'Axis function not implemented' *)
			16#F202:		sTmpText2:=ptrErrorList^.T_LanguagList[21];	(* 'No HDD free resource, time out' *)
			16#F203:		sTmpText2:=ptrErrorList^.T_LanguagList[22];	(* 'HDD error, no file found' *)
			16#F204:		sTmpText2:=ptrErrorList^.T_LanguagList[23];	(* 'Axis Parameter File, wrong syntax' *)
			16#F205:		sTmpText2:=ptrErrorList^.T_LanguagList[26];	(* 'PDOMapping Para File, wrong syntax' *)
			16#F206:		sTmpText2:=ptrErrorList^.T_LanguagList[19];	(* 'Axis function time out error' *)
			16#F207:		sTmpText2:=ptrErrorList^.T_LanguagList[28];	(* 'No Axis Power Supply' *)
			16#F208:		sTmpText2:=ptrErrorList^.T_LanguagList[24];	(* 'Wrong Para Fct: Read Axis Parameter' *)
			16#F209:		sTmpText2:=ptrErrorList^.T_LanguagList[27];	(* 'Wrong Para Fct: Read PDOMapping Parameter' *)
			16#F20A:		sTmpText2:=ptrErrorList^.T_LanguagList[29];	(* 'Wrong Para Fct: Move velocity' *)
			16#F20B:		sTmpText2:=ptrErrorList^.T_LanguagList[31];	(* 'Wrong Para Fct: Move position absolute' *)
			16#F20C:		sTmpText2:=ptrErrorList^.T_LanguagList[32];	(* 'Wrong Para Fct: Move position relative' *)
			16#F20D:	sTmpText2:=ptrErrorList^.T_LanguagList[33];	(* 'Wrong Para Fct: Move referencing' *)
			16#F20E:		sTmpText2:=ptrErrorList^.T_LanguagList[35];	(* 'Wrong Para Fct: Send Axis Parameter' *)
			16#F20F:		sTmpText2:=ptrErrorList^.T_LanguagList[36];	(* 'Wrong Para Fct: Send PDOMapping Parameter' *)
			16#F210:		sTmpText2:=ptrErrorList^.T_LanguagList[37];	(* 'Wrong Para Fct: Master/Slave' *)
			16#F211:		sTmpText2:=ptrErrorList^.T_LanguagList[34];	(* 'Fct CalcAnlgeRefIndex:Ref.Sensor not found' *)
			16#F212:		sTmpText2:=ptrErrorList^.T_LanguagList[30];	(* 'Can not move, no power supply' *)
			16#F213:		sTmpText2:=ptrErrorList^.T_LanguagList[25];	(* 'Limit End Switch Active' *)
			16#F214:		sTmpText2:=ptrErrorList^.T_LanguagList[18];	(* 'ADS communication error' *)
			16#F801:		sTmpText2:=ptrErrorList^.T_LanguagList[1];	(* 'Internal problem, should never appear' *)
			16#F802:		sTmpText2:=ptrErrorList^.T_LanguagList[1];	(* 'Internal problem, should never appear' *)
			16#F803:		sTmpText2:=ptrErrorList^.T_LanguagList[2];	(* 'Antivalence error of the motor encoder' *)
			16#F804:		sTmpText2:=ptrErrorList^.T_LanguagList[3];	(* 'Encoder counter error, >+/- 4 inc' *)
			16#F805:		sTmpText2:=ptrErrorList^.T_LanguagList[4];	(* 'Master encoder X7 counter error, >+/- 4 inc' *)
			16#F806:		sTmpText2:=ptrErrorList^.T_LanguagList[5];	(* 'Heat sink temperature to high (>80°)' *)
			16#F807:		sTmpText2:=ptrErrorList^.T_LanguagList[6];	(* 'Low voltage (<18V) of the +24V logic supply' *)
			16#F808:		sTmpText2:=ptrErrorList^.T_LanguagList[7];	(* 'High voltage X10 (>180V) of the motor power supply' *)
			16#F809:		sTmpText2:=ptrErrorList^.T_LanguagList[8];	(* 'Low voltage X10 (<24V) of the motor power supply' *)
			16#F80A:		sTmpText2:=ptrErrorList^.T_LanguagList[9];	(* 'Short circuit in the motor phase A' *)
			16#F80B:		sTmpText2:=ptrErrorList^.T_LanguagList[10];	(* 'Short circuit in the motor phase B' *)
			16#F80C:		sTmpText2:=ptrErrorList^.T_LanguagList[11];	(* 'Short circuit of a digital output' *)
			16#F80D:	sTmpText2:=ptrErrorList^.T_LanguagList[12];	(* 'Digital input ENABLE going to low level' *)
			16#F80E:		sTmpText2:=ptrErrorList^.T_LanguagList[13];	(* 'Exceed max. countouring error ' *)
			16#F80F:		sTmpText2:=ptrErrorList^.T_LanguagList[14];	(* 'Rotation speed to high, can not read encoder signal' *)
			16#F810:		sTmpText2:=ptrErrorList^.T_LanguagList[15];	(* 'Can not find the commutation' *)
			16#F811:		sTmpText2:=ptrErrorList^.T_LanguagList[16];	(* 'CAN-Communication broken by Node Guarding' *)
			16#F812:		sTmpText2:=ptrErrorList^.T_LanguagList[17];	(* 'I^2t- Controlling triggered (current limit)' *)
			ELSE
						sTmpText2:=ptrErrorList^.T_LanguagList[38];	(* 'Axis general error' *)
			END_CASE;
		END_IF;
		IF (diErrorNr >= 6000000) AND (diErrorNr < 7000000) THEN
			diTmpErrorNr:=diErrorNr - diTmpDeletePrefix;
			CASE diTmpErrorNr OF
			16#F000:		sTmpText2:=ptrErrorList^.T_LanguagList[45];	(* 'Cyl. Function not implemented' *)
			16#F201:		sTmpText2:=ptrErrorList^.T_LanguagList[46];	(* 'Sensor down not active' *)
			16#F202:		sTmpText2:=ptrErrorList^.T_LanguagList[47];	(* 'Sensor up not active' *)
			ELSE
						sTmpText2:=ptrErrorList^.T_LanguagList[48];	(* 'Cyl. general error' *)
			END_CASE;
		END_IF;
		IF (diErrorNr >= 7000000) AND (diErrorNr < 8000000) THEN
			diTmpErrorNr:=diErrorNr - diTmpDeletePrefix;
			CASE diTmpErrorNr OF
			16#F201:		sTmpText2:=ptrErrorList^.T_LanguagList[39];	(* 'ToolLeft: Wrong configuration or Axis missing' *)
			16#F202:		sTmpText2:=ptrErrorList^.T_LanguagList[40];	(* 'ToolCenter: Wrong configuration or Axis missing' *)
			16#F203:		sTmpText2:=ptrErrorList^.T_LanguagList[41];	(* 'ToolRight: Wrong configuration or Axis missing' *)
			16#F204:		sTmpText2:=ptrErrorList^.T_LanguagList[42];	(* 'ToolFeeder: Wrong configuration or Axis missing' *)
			16#F205:		sTmpText2:=ptrErrorList^.T_LanguagList[43];	(* 'GrindFeeder: Wrong configuration or Axis missing' *)
			ELSE
						sTmpText2:=ptrErrorList^.T_LanguagList[44];	(* 'Cyl. general error' *)
			END_CASE;
		END_IF;
		IF (diErrorNr >= 8000000) AND (diErrorNr < 9000000) THEN
			diTmpErrorNr:=diErrorNr - diTmpDeletePrefix;
			CASE diTmpErrorNr OF
			1:			sTmpText2:=ptrErrorList^.T_LanguagList[60];	(* At least one Axis is busy *)
			2:			sTmpText2:=ptrErrorList^.T_LanguagList[68];
			ELSE
						sTmpText2:=ptrErrorList^.T_LanguagList[61];	(* Undefined Station error *)
			END_CASE;
		END_IF;
		IF (diErrorNr >= 10000000) AND (diErrorNr < 16000000) THEN
			diTmpErrorNr:=diErrorNr - diTmpDeletePrefix;
			CASE diTmpErrorNr OF
			16#F000:		sTmpText2:=ptrErrorList^.T_LanguagList[45];	(* 'Cyl. Function not implemented' *)
			16#F201:		sTmpText2:=ptrErrorList^.T_LanguagList[46];	(* 'Sensor down not active' *)
			16#F202:		sTmpText2:=ptrErrorList^.T_LanguagList[47];	(* 'Sensor up not active' *)
			ELSE
						sTmpText2:=ptrErrorList^.T_LanguagList[48];	(* 'Cyl. general error' *)
			END_CASE;
		END_IF;

		sTmpErrorText:=CONCAT(sTmpText1,sTmpText2);
		IF (iCounterLanguage = 1) THEN sErrorTextEnglish:=sTmpErrorText;	END_IF;
		IF (iCounterLanguage = 2) THEN sErrorTextDeutsch:=sTmpErrorText;	END_IF;
		IF (iCounterLanguage = 3) THEN sErrorTextFrancais:=sTmpErrorText;	END_IF;
	END_IF;
END_FOR;
END_FUNCTION_BLOCK

(* POU GENERAL/FB_CHECKACTIVEMOVEMENT, ST *)
FUNCTION_BLOCK FB_CHECKACTIVEMOVEMENT
VAR_INPUT
	T_TwinSafeOut:ST_TWINSAFE_OUT;		(* Output of the TwinSafe components *)
	xKeySwitch:BOOL;							(* Activation and deactivation of the key switch *)
	xBlockChecking:BOOL;						(* block the checking of the axis movement *)
END_VAR
VAR_IN_OUT
	xReset:BOOL;							(* Reset the FB *)
	T_Visu:ST_QVIS;							(* Data structure of the visualisation *)
	T_Station:ST_STATION;					(* Data structure of the station level *)
	T_Process : ST_PROCESS;				(* Data structure of the process level *)
END_VAR
VAR_OUTPUT
	xActiveSetupLevel: BOOL;					(* state of the setuplevel, if it is active *)
	xActiveProcess: BOOL;						(* state of a process if it is active *)
	xActiveStation: BOOL;						(* state of the stationlevel if it is active *)
	xActiveHWStation: BOOL;					(* state of the hardware of the station, if it is active *)
END_VAR
VAR
	xActivateOverlayMessage: BOOL;
	xDoNotCheckMovement: BOOL;
	FallingEdgeKeySwitchOff: F_TRIG;
	iStepSwitchMachineLevel: INT;
	TONWaitTimeStateMachine: TON;
	xPowerSupplyActive: BOOL;
	xTmp: BOOL;
	xStopAxisWithStationFunction: BOOL;
END_VAR
(****************************************************************************************************************************************************)
(*****        This Functionblock check the general movement of all axes. This will be need by change from the station level        ****)
(*****        to the machine level. If case of a change from the station level to the machine level and a axis move than the             ****)
(*****        movement will be stopp																			       ****)
(****************************************************************************************************************************************************)
(* Check Active movement and block visu if active *)
	xTmp:=	(T_Visu.ptrT_ExchgParam^.T_SafetyCtrl.bStateAutoGeometry = 2) OR
			(T_Visu.ptrT_ExchgParam^.T_SafetyCtrl.bStateAutoGroove = 2) OR
			(T_Visu.ptrT_ExchgParam^.T_SafetyCtrl.bStateReference = 2) OR
			(T_Visu.ptrT_ExchgParam^.T_SafetyCtrl.bStateToolCalibration = 2) OR
			(T_Visu.ptrT_ExchgParam^.T_SafetyCtrl.bStateToolTorque = 2) OR
			(T_Visu.ptrT_ExchgParam^.T_SafetyCtrl.bStateTeachInToolLeft = 2) OR
			(T_Visu.ptrT_ExchgParam^.T_SafetyCtrl.bStateTeachInToolCenter = 2) OR
			(T_Visu.ptrT_ExchgParam^.T_SafetyCtrl.bStateTeachInToolRight = 2) OR
			(T_Visu.ptrT_ExchgParam^.T_SafetyCtrl.bStateTeachInToolFeeder = 2) OR
			(T_Visu.ptrT_ExchgParam^.T_SafetyCtrl.bStateTeachInGrindFeeder = 2) OR
			(T_Visu.ptrT_ExchgParam^.T_StationCommon.iWireFeederRefIndexState = 2);
	IF xTmp THEN
		T_StartUp.T_State.xBlockVisuNavigation:=TRUE;	(* Lock the navigation of the visu *)
	END_IF;
	IF T_StartUp.T_State.xBlockVisuNavigation AND NOT(T_StartUp.T_State.xBlockChangeMovementVisu) AND NOT(T_Visu.ptrT_ExchgParam^.T_SafetyCtrl.xBlockVisuObject) AND NOT(xTmp) THEN
		T_StartUp.T_State.xBlockVisuNavigation:=FALSE;	(* Unlock the navigation of the visu *)
	END_IF;

(* Check Setup Level with active key switch and an active movement *)
	IF xReset THEN
		xReset:=FALSE;
		xActivateOverlayMessage:=FALSE;
	END_IF;
	IF NOT(xActivateOverlayMessage) THEN
		xActiveSetupLevel:=	(T_Visu.ptrT_ExchgParam^.T_Visu.bActivSpecialLayer <> 0) AND
							T_StartUp.T_State.xCompleted AND NOT(T_StartUp.T_State.xBlockChangeMovementVisu);
		xDoNotCheckMovement:=	NOT(T_Process.xEnd) AND NOT(T_Process.xError) AND ((T_Process.iFunctNr = 10) OR (T_Process.iFunctNr = 20) OR (T_Process.iFunctNr = 30));
		xActiveProcess:=		NOT(T_Process.xEnd) AND NOT(T_Process.xError) AND (T_Process.iFunctNr = 40);
		xActiveStation:=		NOT(T_Station.TControl.xEnd) AND NOT(T_Station.TControl.xError) AND NOT(xActiveProcess) AND NOT(xDoNotCheckMovement);
		xActiveHWStation:=	T_Station.TControl.xActiveMovement AND NOT(xActiveProcess) AND NOT(xActiveStation) AND NOT(xDoNotCheckMovement);
		(* check if the ToolTorque was activatet *)
		xStopAxisWithStationFunction:=FALSE;
		IF xActiveHWStation THEN
			IF (T_Visu.T_PlcParam.dwActualPage = 220) THEN
				xActiveHWStation:=FALSE;
				xStopAxisWithStationFunction:=TRUE;
			END_IF;
		END_IF;
	END_IF;
	FallingEdgeKeySwitchOff(CLK:=xKeySwitch);
	IF xActiveSetupLevel THEN
		IF FallingEdgeKeySwitchOff.Q THEN
			IF xActiveProcess OR xActiveStation OR xActiveHWStation OR xStopAxisWithStationFunction THEN
				xActivateOverlayMessage:=TRUE;
				iStepSwitchMachineLevel:=1;
			END_IF;
		END_IF;
	END_IF;
(*
	IF NOT(xBlockChecking) THEN
		xActivateOverlayMessage:= xActivateOverlayMessage AND NOT
								(T_Station.TControl.xSecurityCircuitOff OR T_Station.TControl.xSecurityCircuitOn);
	END_IF;
*)
	IF xActivateOverlayMessage THEN
		CASE iStepSwitchMachineLevel OF
		1:	TONWaitTimeStateMachine(IN:=FALSE);
			(* next step *)
			iStepSwitchMachineLevel:=10;
		10:	TONWaitTimeStateMachine(IN:=TRUE,PT:=T#150ms);
			IF TONWaitTimeStateMachine.Q THEN
				TONWaitTimeStateMachine(IN:=FALSE);
				(* next step *)
				iStepSwitchMachineLevel:=20;
			END_IF;
		20:	IF T_TwinSafeOut.QxContactor_K3 AND T_TwinSafeOut.QxContactor_K4 THEN
				xPowerSupplyActive:=TRUE;
				T_Visu.ptrT_ExchgParam^.T_Visu.T_Message.iState:=121;	(* Display message -> The Movement of the machine will be breaked! *)
				(* with switching off of the key switch the power supply is not switched off and the movement are still active *)
				IF xActiveProcess THEN
					T_Process.xStop:=TRUE;
					iStepSwitchMachineLevel:=30;
				END_IF;
				IF xActiveStation THEN
					T_Station.TControl.xStop:=TRUE;
					iStepSwitchMachineLevel:=40;
				END_IF;
				IF xActiveHWStation THEN
					iStepSwitchMachineLevel:=60;
				END_IF;
				IF xStopAxisWithStationFunction THEN
					iStepSwitchMachineLevel:=70;
				END_IF;
			ELSE
				(* with switching off of the key switch the power supply is switched off *)
				xPowerSupplyActive:=FALSE;
				(* next step *)
				iStepSwitchMachineLevel:=80;
			END_IF;
		30:	IF T_Process.xEnd THEN
				(* next step *)
				iStepSwitchMachineLevel:=80;
			END_IF;
			IF NOT(T_TwinSafeOut.QxContactor_K3) OR NOT(T_TwinSafeOut.QxContactor_K4) THEN
				xPowerSupplyActive:=FALSE;
				iStepSwitchMachineLevel:=80;
			END_IF;
			T_Visu.ptrT_ExchgParam^.T_Visu.T_Message.iState:=121;	(* Display message -> The Movement of the machine will be breaked! *)
		40:	IF T_Station.TControl.xEnd THEN
				(* next step *)
				T_Station.TControl.xStop:=FALSE;
				iStepSwitchMachineLevel:=60;
			END_IF;
			IF NOT(T_TwinSafeOut.QxContactor_K3) OR NOT(T_TwinSafeOut.QxContactor_K4) THEN
				xPowerSupplyActive:=FALSE;
				iStepSwitchMachineLevel:=80;
			END_IF;
			T_Visu.ptrT_ExchgParam^.T_Visu.T_Message.iState:=121;	(* Display message -> The Movement of the machine will be breaked! *)
		60:	IF T_Station.THardware.TAxisToolLeft.T_CtrleSingle.xDone AND NOT(T_Station.THardware.TAxisToolLeft.T_CtrleSingle.xErr) THEN
				T_Station.THardware.TAxisToolLeft.T_CtrleSingle.iFunction:=5;
				T_Station.THardware.TAxisToolLeft.T_CtrleSingle.xExecute:=TRUE;
			END_IF;
			IF NOT(T_Station.THardware.TAxisToolLeft.T_CtrleSingle.xDone) AND T_Station.THardware.TAxisToolLeft.T_CtrleSingle.xNotMoving AND NOT(T_Station.THardware.TAxisToolLeft.T_CtrleSingle.xErr) THEN
				T_Station.THardware.TAxisToolLeft.T_CtrleSingle.xReset:=TRUE;
			END_IF;
			IF T_Station.THardware.TAxisToolRight.T_CtrleSingle.xDone AND NOT(T_Station.THardware.TAxisToolRight.T_CtrleSingle.xErr) THEN
				T_Station.THardware.TAxisToolRight.T_CtrleSingle.iFunction:=5;
				T_Station.THardware.TAxisToolRight.T_CtrleSingle.xExecute:=TRUE;
			END_IF;
			IF NOT(T_Station.THardware.TAxisToolRight.T_CtrleSingle.xDone) AND T_Station.THardware.TAxisToolRight.T_CtrleSingle.xNotMoving AND NOT(T_Station.THardware.TAxisToolRight.T_CtrleSingle.xErr) THEN
				T_Station.THardware.TAxisToolRight.T_CtrleSingle.xReset:=TRUE;
			END_IF;
			IF T_Station.THardware.TAxisToolCenter.T_CtrleSingle.xDone AND NOT(T_Station.THardware.TAxisToolCenter.T_CtrleSingle.xErr) THEN
				T_Station.THardware.TAxisToolCenter.T_CtrleSingle.iFunction:=5;
				T_Station.THardware.TAxisToolCenter.T_CtrleSingle.xExecute:=TRUE;
			END_IF;
			IF NOT(T_Station.THardware.TAxisToolCenter.T_CtrleSingle.xDone) AND T_Station.THardware.TAxisToolCenter.T_CtrleSingle.xNotMoving AND NOT(T_Station.THardware.TAxisToolCenter.T_CtrleSingle.xErr) THEN
				T_Station.THardware.TAxisToolCenter.T_CtrleSingle.xReset:=TRUE;
			END_IF;
			IF T_Station.THardware.TAxisToolFeeder.T_CtrleSingle.xDone AND NOT(T_Station.THardware.TAxisToolFeeder.T_CtrleSingle.xErr) THEN
				T_Station.THardware.TAxisToolFeeder.T_CtrleSingle.iFunction:=5;
				T_Station.THardware.TAxisToolFeeder.T_CtrleSingle.xExecute:=TRUE;
			END_IF;
			IF NOT(T_Station.THardware.TAxisToolFeeder.T_CtrleSingle.xDone) AND NOT(T_Station.THardware.TAxisToolFeeder.T_CtrleSingle.xNotMoving) AND NOT(T_Station.THardware.TAxisToolFeeder.T_CtrleSingle.xErr) THEN
				T_Station.THardware.TAxisToolFeeder.T_CtrleSingle.iFunction:=5;
				T_Station.THardware.TAxisToolFeeder.T_CtrleSingle.xExecute:=TRUE;
			END_IF;
			IF NOT(T_Station.THardware.TAxisToolFeeder.T_CtrleSingle.xDone) AND T_Station.THardware.TAxisToolFeeder.T_CtrleSingle.xNotMoving AND NOT(T_Station.THardware.TAxisToolFeeder.T_CtrleSingle.xErr) THEN
				T_Station.THardware.TAxisToolFeeder.T_CtrleSingle.xReset:=TRUE;
			END_IF;
			IF T_Station.THardware.TAxisGrindFeeder.T_CtrleSingle.xDone AND NOT(T_Station.THardware.TAxisGrindFeeder.T_CtrleSingle.xErr) THEN
				T_Station.THardware.TAxisGrindFeeder.T_CtrleSingle.iFunction:=5;
				T_Station.THardware.TAxisGrindFeeder.T_CtrleSingle.xExecute:=TRUE;
			END_IF;
			IF NOT(T_Station.THardware.TAxisGrindFeeder.T_CtrleSingle.xDone) AND NOT(T_Station.THardware.TAxisGrindFeeder.T_CtrleSingle.xNotMoving) AND NOT(T_Station.THardware.TAxisGrindFeeder.T_CtrleSingle.xErr) THEN
				T_Station.THardware.TAxisGrindFeeder.T_CtrleSingle.iFunction:=5;
				T_Station.THardware.TAxisGrindFeeder.T_CtrleSingle.xExecute:=TRUE;
			END_IF;
			IF NOT(T_Station.THardware.TAxisGrindFeeder.T_CtrleSingle.xDone) AND T_Station.THardware.TAxisGrindFeeder.T_CtrleSingle.xNotMoving AND NOT(T_Station.THardware.TAxisGrindFeeder.T_CtrleSingle.xErr) THEN
				T_Station.THardware.TAxisGrindFeeder.T_CtrleSingle.xReset:=TRUE;
			END_IF;
			IF NOT(T_Station.THardware.TCylToolTension.T_CtrleCyl.xDone) THEN T_Station.THardware.TCylToolTension.T_CtrleCyl.xReset:=TRUE; END_IF;
			T_Visu.ptrT_ExchgParam^.T_Visu.T_Message.iState:=121;	(* Display message -> The Movement of the machine will be breaked! *)
			(* next step *)
			iStepSwitchMachineLevel:=80;
		70:	IF T_Station.TControl.xEnd THEN
				(* next step *)
				T_Station.TControl.iFunctNr:=3;
				T_Station.TControl.xStart:=TRUE;
				iStepSwitchMachineLevel:=71;
			END_IF;
			IF NOT(T_TwinSafeOut.QxContactor_K3) OR NOT(T_TwinSafeOut.QxContactor_K4) THEN
				xPowerSupplyActive:=FALSE;
				iStepSwitchMachineLevel:=80;
			END_IF;
			T_Visu.ptrT_ExchgParam^.T_Visu.T_Message.iState:=121;	(* Display message -> The Movement of the machine will be breaked! *)
		71:	IF NOT(T_Station.TControl.xStart) AND T_Station.TControl.xEnd THEN
				(* next step *)
				iStepSwitchMachineLevel:=80;
			END_IF;
			IF NOT(T_TwinSafeOut.QxContactor_K3) OR NOT(T_TwinSafeOut.QxContactor_K4) THEN
				xPowerSupplyActive:=FALSE;
				iStepSwitchMachineLevel:=80;
			END_IF;
		80:	IF NOT(T_Visu.T_CtrleVisu.xExecute) AND T_Visu.T_CtrleVisu.xDone THEN
				T_Visu.ptrT_ExchgParam^.T_Visu.T_Message.iState:=0;
				T_Visu.ptrT_ExchgParam^.T_Visu.bActivSpecialLayer:=0;
				T_Visu.ptrT_ExchgParam^.T_TouchScreenBtPanel.iStateBtLeft:=0;
				T_Visu.ptrT_ExchgParam^.T_TouchScreenNavPanel.wState:=1;
				T_Visu.T_PlcParam.dwSetNewPage:=16#A;	(* Main Page wird aufgerufen *)
				T_Visu.T_CtrleVisu.iFunction:=1;
				T_Visu.T_CtrleVisu.xExecute:=TRUE;
				iStepSwitchMachineLevel:=90;
			END_IF;
		90:	IF NOT(T_Visu.T_CtrleVisu.xExecute) AND T_Visu.T_CtrleVisu.xDone THEN
				T_StartUp.T_State.xBlockChangeMovementVisu:=TRUE;	(* Lock the navigation of the visu *)
				T_Visu.ptrT_ExchgParam^.T_SafetyCtrl.xBlockVisuObject:=TRUE;
				T_StartUp.T_State.xBlockVisuNavigation:=FALSE;	(* Unlock the navigation of the visu *)
				T_Visu.ptrT_ExchgParam^.T_SafetyCtrl.bStateAutoGeometry:=1;
				T_Visu.ptrT_ExchgParam^.T_SafetyCtrl.bStateAutoGroove:=1;
				T_Visu.ptrT_ExchgParam^.T_SafetyCtrl.bStateReference:=1;
				T_Visu.ptrT_ExchgParam^.T_SafetyCtrl.bStateToolCalibration:=1;
				T_Visu.ptrT_ExchgParam^.T_SafetyCtrl.bStateToolTorque:=1;
				T_Visu.ptrT_ExchgParam^.T_SafetyCtrl.bStateTeachInToolLeft:=1;
				T_Visu.ptrT_ExchgParam^.T_SafetyCtrl.bStateTeachInToolCenter:=1;
				T_Visu.ptrT_ExchgParam^.T_SafetyCtrl.bStateTeachInToolRight:=1;
				T_Visu.ptrT_ExchgParam^.T_SafetyCtrl.bStateTeachInToolFeeder:=1;
				T_Visu.ptrT_ExchgParam^.T_SafetyCtrl.bStateTeachInGrindFeeder:=1;
				T_Visu.ptrT_ExchgParam^.T_StationCommon.iWireFeederRefIndexState:=1;
				(* Overlay Message Error *)
				T_Visu.ptrT_ExchgParam^.T_SafetyCtrl.bStateMessageError:=1;
				T_Visu.ptrT_ExchgParam^.T_SafetyCtrl.bStateMessageInfo:=0;
				T_Visu.ptrT_ExchgParam^.T_SafetyCtrl.bStateMessageWarning:=0;
				IF xPowerSupplyActive THEN
					T_Visu.ptrT_ExchgParam^.T_SafetyCtrl.iMsgErrorLine1:=18;	(* WHILE A MOVEMENT THE KEY SWITCH *)
					T_Visu.ptrT_ExchgParam^.T_SafetyCtrl.iMsgErrorLine2:=18;	(* HAS BEEN SWITCHED OFF! *)
					T_Visu.ptrT_ExchgParam^.T_SafetyCtrl.iMsgErrorLine3:=18;	(* NOW YOU ARE ON THE NORMAL OPERATION *)
					T_Visu.ptrT_ExchgParam^.T_SafetyCtrl.iMsgErrorLine4:=18;	(* AND THE POWER SUPPLY IS STILL SWITCHED ON *)
					T_Visu.ptrT_ExchgParam^.T_SafetyCtrl.xConfirmMsgError:=FALSE;
				ELSE
					T_Visu.ptrT_ExchgParam^.T_SafetyCtrl.iMsgErrorLine1:=17;	(* WHILE A MOVEMENT THE KEY SWITCH *)
					T_Visu.ptrT_ExchgParam^.T_SafetyCtrl.iMsgErrorLine2:=17;	(* HAS BEEN SWITCHED OFF! *)
					T_Visu.ptrT_ExchgParam^.T_SafetyCtrl.iMsgErrorLine3:=17;	(* NOW YOU ARE ON THE NORMAL OPERATION *)
					T_Visu.ptrT_ExchgParam^.T_SafetyCtrl.iMsgErrorLine4:=17;	(* AND THE POWER SUPPLY IS SWITCHED OFF *)
					T_Visu.ptrT_ExchgParam^.T_SafetyCtrl.xConfirmMsgError:=FALSE;
				END_IF;
				(* next step *)
				iStepSwitchMachineLevel:=100;
			END_IF;
		100:	IF T_Visu.ptrT_ExchgParam^.T_SafetyCtrl.xConfirmMsgError THEN
				T_StartUp.T_State.xBlockChangeMovementVisu:=FALSE;	(* Unlock the navigation of the visu *)
				T_Visu.ptrT_ExchgParam^.T_SafetyCtrl.xBlockVisuObject:=FALSE;
				T_StartUp.T_State.xBlockVisuNavigation:=FALSE;	(* Unlock the navigation of the visu *)
				T_Visu.ptrT_ExchgParam^.T_SafetyCtrl.bStateAutoGeometry:=1;
				T_Visu.ptrT_ExchgParam^.T_SafetyCtrl.bStateAutoGroove:=1;
				T_Visu.ptrT_ExchgParam^.T_SafetyCtrl.bStateReference:=1;
				T_Visu.ptrT_ExchgParam^.T_SafetyCtrl.bStateToolCalibration:=1;
				T_Visu.ptrT_ExchgParam^.T_SafetyCtrl.bStateToolTorque:=1;
				T_Visu.ptrT_ExchgParam^.T_SafetyCtrl.bStateTeachInToolLeft:=1;
				T_Visu.ptrT_ExchgParam^.T_SafetyCtrl.bStateTeachInToolCenter:=1;
				T_Visu.ptrT_ExchgParam^.T_SafetyCtrl.bStateTeachInToolRight:=1;
				T_Visu.ptrT_ExchgParam^.T_SafetyCtrl.bStateTeachInToolFeeder:=1;
				T_Visu.ptrT_ExchgParam^.T_SafetyCtrl.bStateTeachInGrindFeeder:=1;
				T_Visu.ptrT_ExchgParam^.T_StationCommon.iWireFeederRefIndexState:=1;
				T_Visu.ptrT_ExchgParam^.T_SafetyCtrl.bStateMessageError:=0;
				T_Visu.ptrT_ExchgParam^.T_SafetyCtrl.xConfirmMsgError:=FALSE;
				xActivateOverlayMessage:=FALSE;
				iStepSwitchMachineLevel:=1;
			END_IF;
			IF NOT(T_TwinSafeOut.QxContactor_K3) OR NOT(T_TwinSafeOut.QxContactor_K4) THEN
				T_Visu.ptrT_ExchgParam^.T_SafetyCtrl.iMsgErrorLine1:=17;	(* WHILE A MOVEMENT THE KEY SWITCH *)
				T_Visu.ptrT_ExchgParam^.T_SafetyCtrl.iMsgErrorLine2:=17;	(* HAS BEEN SWITCHED OFF! *)
				T_Visu.ptrT_ExchgParam^.T_SafetyCtrl.iMsgErrorLine3:=17;	(* NOW YOU ARE ON THE NORMAL OPERATION *)
				T_Visu.ptrT_ExchgParam^.T_SafetyCtrl.iMsgErrorLine4:=17;	(* AND THE POWER SUPPLY IS SWITCHED OFF *)
			END_IF;
			IF T_TwinSafeOut.QxContactor_K3 AND T_TwinSafeOut.QxContactor_K4  THEN
				T_Visu.ptrT_ExchgParam^.T_SafetyCtrl.iMsgErrorLine1:=18;	(* WHILE A MOVEMENT THE KEY SWITCH *)
				T_Visu.ptrT_ExchgParam^.T_SafetyCtrl.iMsgErrorLine2:=18;	(* HAS BEEN SWITCHED OFF! *)
				T_Visu.ptrT_ExchgParam^.T_SafetyCtrl.iMsgErrorLine3:=18;	(* NOW YOU ARE ON THE NORMAL OPERATION *)
				T_Visu.ptrT_ExchgParam^.T_SafetyCtrl.iMsgErrorLine4:=18;	(* AND THE POWER SUPPLY IS STILL SWITCHED ON *)
			END_IF;
		END_CASE;
	END_IF;
END_FUNCTION_BLOCK

(* POU PRG_VISU_LAYER5/PRG_VISU, FBD *)
PROGRAM PRG_VISU
VAR
	fbVisuQVis: FBQVIS;
	xSecurityKey: BOOL;
	FBCtrleButton: FB_CTRLEBUTTON;
END_VAR
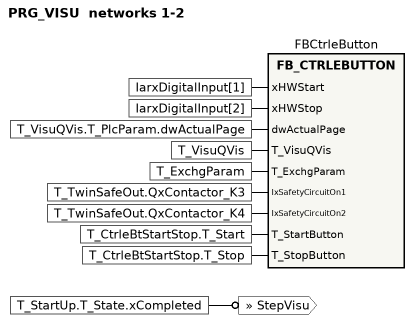
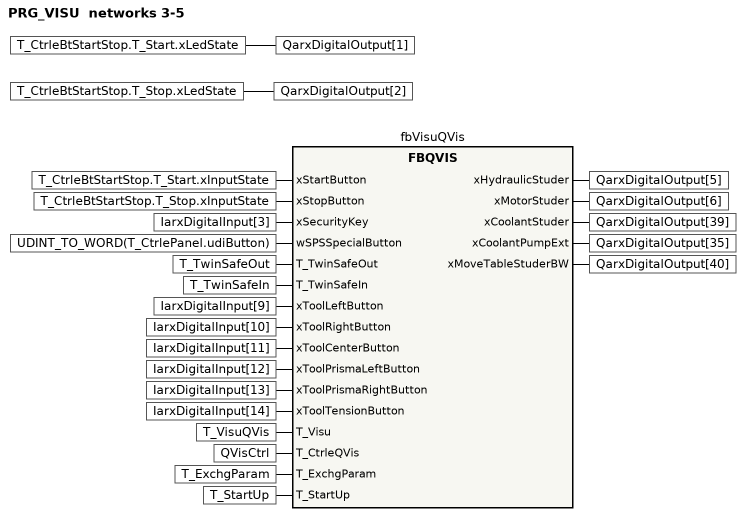
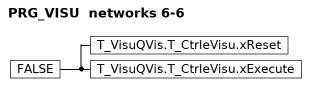
_FBD_ (* Function Block Diagram *)
NETWORK 1 (* VISUALISATION LEVEL-->LAYER 5 *)
	FBCtrleButton:FB_CTRLEBUTTON(xHWStart: IarxDigitalInput[1], xHWStop: IarxDigitalInput[2], dwActualPage: T_VisuQVis.T_PlcParam.dwActualPage, T_VisuQVis: T_VisuQVis, T_ExchgParam: T_ExchgParam, IxSafetyCircuitOn1: T_TwinSafeOut.QxContactor_K3, IxSafetyCircuitOn2: T_TwinSafeOut.QxContactor_K4, T_StartButton: T_CtrleBtStartStop.T_Start, T_StopButton: T_CtrleBtStartStop.T_Stop)
NETWORK 2
	NOT T_StartUp.T_State.xCompleted => >>StepVisu
NETWORK 3
	T_CtrleBtStartStop.T_Start.xLedState => QarxDigitalOutput[1]
NETWORK 4
	T_CtrleBtStartStop.T_Stop.xLedState => QarxDigitalOutput[2]
NETWORK 5 StepVisu:
	fbVisuQVis:FBQVIS(xStartButton: T_CtrleBtStartStop.T_Start.xInputState, xStopButton: T_CtrleBtStartStop.T_Stop.xInputState, xSecurityKey: IarxDigitalInput[3], wSPSSpecialButton: UDINT_TO_WORD(T_CtrlePanel.udiButton), T_TwinSafeOut: T_TwinSafeOut, T_TwinSafeIn: T_TwinSafeIn, xToolLeftButton: IarxDigitalInput[9], xToolRightButton: IarxDigitalInput[10], xToolCenterButton: IarxDigitalInput[11], xToolPrismaLeftButton: IarxDigitalInput[12], xToolPrismaRightButton: IarxDigitalInput[13], xToolTensionButton: IarxDigitalInput[14], T_Visu: T_VisuQVis, T_CtrleQVis: QVisCtrl, T_ExchgParam: T_ExchgParam, T_StartUp: T_StartUp, xMotorStuder => QarxDigitalOutput[6], xCoolantStuder => QarxDigitalOutput[39], xCoolantPumpExt => QarxDigitalOutput[35], xMoveTableStuderBW => QarxDigitalOutput[40]) => QarxDigitalOutput[5]
NETWORK 6
	FALSE => T_VisuQVis.T_CtrleVisu.xReset, T_VisuQVis.T_CtrleVisu.xExecute
_END_FBD_
(* the same logic as Structured Text *)
(* Network 1: VISUALISATION LEVEL-->LAYER 5 *)
FBCtrleButton(xHWStart := IarxDigitalInput[1], xHWStop := IarxDigitalInput[2], dwActualPage := T_VisuQVis.T_PlcParam.dwActualPage, T_VisuQVis := T_VisuQVis, T_ExchgParam := T_ExchgParam, IxSafetyCircuitOn1 := T_TwinSafeOut.QxContactor_K3, IxSafetyCircuitOn2 := T_TwinSafeOut.QxContactor_K4, T_StartButton := T_CtrleBtStartStop.T_Start, T_StopButton := T_CtrleBtStartStop.T_Stop);
(* Network 2 *)
IF NOT T_StartUp.T_State.xCompleted THEN JMP StepVisu; END_IF;
(* Network 3 *)
QarxDigitalOutput[1] := T_CtrleBtStartStop.T_Start.xLedState;
(* Network 4 *)
QarxDigitalOutput[2] := T_CtrleBtStartStop.T_Stop.xLedState;
(* Network 5 *)
StepVisu:
fbVisuQVis(xStartButton := T_CtrleBtStartStop.T_Start.xInputState, xStopButton := T_CtrleBtStartStop.T_Stop.xInputState, xSecurityKey := IarxDigitalInput[3], wSPSSpecialButton := UDINT_TO_WORD(T_CtrlePanel.udiButton), T_TwinSafeOut := T_TwinSafeOut, T_TwinSafeIn := T_TwinSafeIn, xToolLeftButton := IarxDigitalInput[9], xToolRightButton := IarxDigitalInput[10], xToolCenterButton := IarxDigitalInput[11], xToolPrismaLeftButton := IarxDigitalInput[12], xToolPrismaRightButton := IarxDigitalInput[13], xToolTensionButton := IarxDigitalInput[14], T_Visu := T_VisuQVis, T_CtrleQVis := QVisCtrl, T_ExchgParam := T_ExchgParam, T_StartUp := T_StartUp);
QarxDigitalOutput[6] := fbVisuQVis.xMotorStuder;
QarxDigitalOutput[39] := fbVisuQVis.xCoolantStuder;
QarxDigitalOutput[35] := fbVisuQVis.xCoolantPumpExt;
QarxDigitalOutput[40] := fbVisuQVis.xMoveTableStuderBW;
QarxDigitalOutput[5] := fbVisuQVis.xHydraulicStuder;
(* Network 6 *)
T_VisuQVis.T_CtrleVisu.xReset := FALSE;
T_VisuQVis.T_CtrleVisu.xExecute := FALSE;
END_PROGRAM

(* POU PRG_VISU_LAYER5/FB_VISU/FBQVIS, ST *)
FUNCTION_BLOCK FBQVIS
VAR_INPUT
	xStartButton:BOOL;					(* external start button *)
	xStopButton:BOOL;					(* external stop button *)
	xSecurityKey:BOOL;					(* state of the keyswitch *)
	wSPSSpecialButton:WORD;			(* input of the special button of the controlpanel *)
	T_TwinSafeOut:ST_TWINSAFE_OUT;	(* Output of the TwinSAFE components *)
	T_TwinSafeIn:ST_TWINSAFE_IN;		(* Input of the TwinSAFE components *)
(*22.12.2009: KFS	{	*)
	xToolLeftButton:BOOL;					(* Signal of the button for closing the ToolLeft-->this is only for the MicroRod *)
	xToolRightButton:BOOL;				(* Signal of the button for closing the ToolRight-->this is only for the MicroRod *)
	xToolCenterButton:BOOL;				(* Signal of the button for closing the ToolCenter-->this is only for the MicroRod *)
	xToolPrismaLeftButton:BOOL;			(* Signal of the button for closing the ToolPrismaLeft-->this is only for the MicroRod *)
	xToolPrismaRightButton:BOOL;			(* Signal of the button for closing the ToolPrismaRight-->this is only for the MicroRod *)
	xToolTensionButton:BOOL;				(* Signal of the button for activate the ToolTension-->this is only for the MicroRod *)
(*22.12.2009: KFS	}	*)
END_VAR
VAR_OUTPUT
(* SOA 02.02.2023     {     *)
	xHydraulicStuder: 	BOOL;  					(*Hydraulic Pump of Studer S20 Machine*)
	xMotorStuder: BOOL;						(*Grinding-Engine of Studer S20 Machine*)
	xCoolantStuder: BOOL;						(*Coolant Pump of Studer S20 Machine*)
	xCoolantPumpExt: BOOL;					(*Coolant Pump external*)
	xMoveTableStuderBW:BOOL;
(* SOA 02.02.2023    }   *)
END_VAR
VAR_IN_OUT
	T_Visu:ST_QVIS;
	T_CtrleQVis:ST_QVISCTRLE;
	T_ExchgParam:ST_QVIS_EXCHG_PARAM;
	T_StartUp:ST_STARTUP;
END_VAR
VAR
	RisingEdgeActiv:R_TRIG;
	RisingEdgeExecute:R_TRIG;
	RisingEdgeExecuteAction:R_TRIG;
	RisingEdgeBtPanelLeft:R_TRIG;
	FallingEdgeBtPanelLeft:F_TRIG;
	RisingEdgeSpecialLayer:R_TRIG;
	FallingEdgeSpecialLayer:F_TRIG;
	RisingEdgeTouchScreenNavPanel:R_TRIG;
	FallingEdgeTouchScreenNavPanel:F_TRIG;
	RisingEdgeBtPanelRight:R_TRIG;
	FallingEdgeBtPanelRight:F_TRIG;
	RisingEdgeBtFunctionPanel:R_TRIG;
	FallingEdgeBtFunctionPanel:F_TRIG;
	RisingEdgeDynPassword:R_TRIG;
	RisingEdgeGeometryManagement:R_TRIG;
	RisingEdgeToolDiameter:R_TRIG;
	RisingEdgePrisma:R_TRIG;
	xChangePage:BOOL:=FALSE;
	dwInCount_QVisCmd:DWORD:=0;
	xTmp: BOOL;
	wActivBtLeft: WORD;
	wActivBtRight: WORD;
	fbQvisInitPage:FBQVIS_INITPAGE;
	xNavPanelChangePage: BOOL;
	xBtPanelLeftChangePage:BOOL;
	xBtPanelRightChangePage: BOOL; (*SOA*)
	xNextPageVertical:BOOL;
	xSetParameterPage:BOOL;
	xActivationSection1: BOOL;
	xActivationSection2: BOOL;
	xActivationSection3: BOOL;
	xActivationSection4: BOOL;
	xActivationSection5: BOOL; (*SOA *)
	xActivationSection6: BOOL; (*SOA *)

	xSetPitchEqual: BOOL;
	iStepAction: INT;
	xStepActionDone: BOOL;
	bOldActivSpecialLayer: BYTE;
	wSpecialLayerGeneralActivTask: WORD;
	wSpecialLayerToolRotActivTask: WORD;
	wSpecialLayerWireFeedActivTask: WORD;
	wSpecialLayerGrindAxisActivTask: WORD;
	wSpecialLayerGeneralActivPage: WORD;
	wSpecialLayerToolRotActivPage: WORD;
	wSpecialLayerWireFeedActivPage: WORD;
	wSpecialLayerGrindAxisActivPage: WORD;
	dwSetNewPage: DWORD;
	wNormalLayerActivTask: WORD;
	wNormalLayerActivPage: WORD;
	ii: INT;
	wTmp: WORD;
	awNormalLayerActivPage:ARRAY [1..6] OF WORD;
	awSpecialLayerGeneralActivPage:ARRAY [1..6] OF WORD;
	awSpecialLayerToolRotActivPage:ARRAY [1..6] OF WORD;
	awSpecialLayerWireFeedActivPage:ARRAY [1..6] OF WORD;
	awSpecialLayerGrindAxisActivPage:ARRAY [1..6] OF WORD;
	wTmpNormalLayerActivTask: WORD;
	wTmpSpecialLayerGeneralActivTask: WORD;
	wTmpSpecialLayerToolRotActivTask: WORD;
	wTmpSpecialLayerWireFeedActivTask: WORD;
	wTmpSpecialLayerGrindAxisActivTask: WORD;
	wStandardPageNr: WORD;
	iTmpActivBtLeft: INT;
	(* Random *)
	fbGetCpuAccount:GETCPUCOUNTER;
	fbPwSystem:FBPW_SYSTEM;
	(* Pw *)
	iPwSystem:INT;
	iStepCounter: INT;
	arSaveToolGeometry:ST_GEOMETRY;
	rSectionPitch: REAL;
	ptxActiveSection1: POINTER TO BOOL;
	ptxActiveSection2: POINTER TO BOOL;
	ptxActiveSection3: POINTER TO BOOL;
	ptxActiveSection4: POINTER TO BOOL;
	ptxActiveSection5: POINTER TO BOOL;
	ptxActiveSection6: POINTER TO BOOL;

	xOverlayMeasureToolDia: BOOL;
	xPlungeActivation: BOOL;
	xDisplaceActivation: BOOL;
	xCorrectionToolDiameterAdd: BOOL;
	xCorrectionToolDiameterAddMore: BOOL;
	xCorrectionToolDiameterSub: BOOL;
	xCorrectionToolDiameterSubMore: BOOL;
	xResetToolDiameterCorrection: BOOL;
	xKeyPadActivation: BOOL;
	xFctCorrectionToolDiameter: BOOL;
	rCorrectionValue: REAL;

(* Key panel button "Esc"/"Enter" *)
	RisingEdgeKeyPanel_Esc:R_TRIG;
	RisingEdgeKeyPanel_Enter:R_TRIG;
(*22.12.2009: KFS	{	 *)
(* External button for the tool-clamping*)
	RisingEdgeBtToolLeft:R_TRIG;
	RisingEdgeBtToolRight:R_TRIG;
	RisingEdgeBtToolCenter:R_TRIG;
	RisingEdgeBtToolPrismaLeft:R_TRIG;
	RisingEdgeBtToolPrismaRight:R_TRIG;
	RisingEdgeBtToolTension:R_TRIG;
(*22.12.2009: KFS	}	 *)
(* variable start action *)
	TimerAction:TON;
	TimerNotReady:TOF;
	tTimeOutAction:TIME;
	xSelectPrisma: BOOL;
	xToolTensForceAdd: BOOL;
	xToolTensForceAddMore: BOOL;
	xToolTensForceSub: BOOL;
	xToolTensForceSubMore: BOOL;
	xResetCalculToolRotTorque: BOOL;
	rCalcTotalToolLength: REAL;
	xTmpSecurityKey: BOOL;
	RisingEdgeTemp:R_TRIG;
	TONWAIT: TON;
	xPart1: BOOL;
	xPart2: BOOL;
	xPart3: BOOL;
	xPart4: BOOL;
	xPart5: BOOL;
	xPart6: BOOL;

	iPartActive: INT;
	xToolRotationMasterSlave: BOOL;
	xSwitchMasterSlave: BOOL;
	xQvisActiv: BOOL;
	TimerQVis: TON;
	RisingEdgeReset:R_TRIG;
	xConfirmResetFB: BOOL;
	xFirstRead: BOOL;
	ptrTeachINAxis:POINTER TO ST_AXIS;
	ptrCylAction:POINTER TO ST_CYLINDER;
	xStopAxis: BOOL;
	xMoveRelPosition: BOOL;
	TParaAxisTeachIN:ST_EXCHG_PARAM_TEACHIN;
	xMoveContinousVel: BOOL;
	xMoveAbsPosition: BOOL;
	bButtonPanelLocked: BYTE;
	xDelayActionBtPanelRight: BOOL;
	TimerPressBtPanelRight: TON;

